LIN {X 0,Y 183.48,Z 465.973,A -85,B 0,C 180,E1 -22041.184,E2 -22041.184} C_VEL
LIN {X 0,Y 183.189,Z 466.318,A -85,B 0,C 180,E1 -22045.596,E2 -22045.596} C_VEL
LIN {X 0,Y 183.308,Z 465.887,A -85,B 0,C 180,E1 -22047.799,E2 -22047.799} C_VEL
LIN {X 0,Y 183.482,Z 465.038,A -85,B 0,C 180,E1 -22049.996,E2 -22049.996} C_VEL
LIN {X 0,Y 183.338,Z 463.763,A -85,B 0,C 180,E1 -22052.193,E2 -22052.193} C_VEL
LIN {X 0,Y 183.267,Z 461.02,A -85,B 0,C 180,E1 -22055.497,E2 -22055.497} C_VEL
LIN {X 0,Y 183.529,Z 457.223,A -85,B 0,C 180,E1 -22058.806,E2 -22058.806} C_VEL
LIN {X 0,Y 184.122,Z 452.262,A -85,B 0,C 180,E1 -22062.114,E2 -22062.114} C_VEL
LIN {X 0,Y 185.268,Z 446.001,A -85,B 0,C 180,E1 -22065.394,E2 -22065.394} C_VEL
LIN {X 0,Y 186.943,Z 438.169,A -85,B 0,C 180,E1 -22068.63,E2 -22068.63} C_VEL
LIN {X 0,Y 188.899,Z 429.24,A -85,B 0,C 180,E1 -22071.543,E2 -22071.543} C_VEL
LIN {X 0,Y 190.919,Z 420.311,A -85,B 0,C 180,E1 -22073.88,E2 -22073.88} C_VEL
LIN {X 0,Y 193.253,Z 409.393,A -85,B 0,C 180,E1 -22076.158,E2 -22076.158} C_VEL
LIN {X 0,Y 195.335,Z 398.733,A -85,B 0,C 180,E1 -22077.88,E2 -22077.88} C_VEL
LIN {X 0,Y 197.244,Z 387.011,A -85,B 0,C 180,E1 -22079.329,E2 -22079.329} C_VEL
LIN {X 0,Y 198.937,Z 373.736,A -85,B 0,C 180,E1 -22080.513,E2 -22080.513} C_VEL
LIN {X 0,Y 199.925,Z 361.7,A -85,B 0,C 180,E1 -22081.225,E2 -22081.225} C_VEL
LIN {X 0,Y 201.881,Z 312.915,A -85,B 0,C 180,E1 -22082.925,E2 -22082.925} C_VEL
LIN {X 0,Y 198.695,Z 281.913,A -85,B 0,C 180,E1 -22084.649,E2 -22084.649} C_VEL
LIN {X 0,Y 191.948,Z 264.141,A -85,B 0,C 180,E1 -22086.507,E2 -22086.507} C_VEL
LIN {X 0,Y 187.121,Z 252.944,A -85,B 0,C 180,E1 -22087.932,E2 -22087.932} C_VEL
LIN {X 0,Y 185.488,Z 246.381,A -85,B 0,C 180,E1 -22091.468,E2 -22091.468} C_VEL
LIN {X 0,Y 185.505,Z 246.376,A -85,B 0,C 180,E1 -22097.003,E2 -22097.003} C_VEL
LIN {X 0,Y 185.519,Z 246.373,A -85,B 0,C 180,E1 -22099.908,E2 -22099.908} C_VEL
LIN {X 0,Y 185.525,Z 246.373,A -85,B 0,C 180,E1 -22102.691,E2 -22102.691} C_VEL
LIN {X 0,Y 185.521,Z 246.373,A -85,B 0,C 180,E1 -22107.97,E2 -22107.97} C_VEL
LIN {X 0,Y 185.559,Z 246.367,A -85,B 0,C 180,E1 -22110.572,E2 -22110.572} C_VEL
LIN {X 0,Y 185.583,Z 246.364,A -85,B 0,C 180,E1 -22115.381,E2 -22115.381} C_VEL
LIN {X 0,Y 185.685,Z 246.348,A -85,B 0,C 180,E1 -22121.098,E2 -22121.098} C_VEL
LIN {X 0,Y 185.696,Z 246.35,A -85,B 0,C 180,E1 -22126.874,E2 -22126.874} C_VEL
LIN {X 0,Y 185.978,Z 246.319,A -85,B 0,C 180,E1 -22131.305,E2 -22131.305} C_VEL
LIN {X 0,Y 186.171,Z 246.257,A -85,B 0,C 180,E1 -22137.836,E2 -22137.836} C_VEL
LIN {X 0,Y 186.367,Z 246.222,A -85,B 0,C 180,E1 -22139.999,E2 -22139.999} C_VEL
LIN {X 0,Y 185.874,Z 246.321,A -85,B 0,C 180,E1 -22144.336,E2 -22144.336} C_VEL
LIN {X 0,Y 185.944,Z 246.321,A -85,B 0,C 180,E1 -22148.695,E2 -22148.695} C_VEL
LIN {X 0,Y 185.684,Z 246.349,A -85,B 0,C 180,E1 -22153.125,E2 -22153.125} C_VEL
LIN {X 0,Y 185.621,Z 246.358,A -85,B 0,C 180,E1 -22157.631,E2 -22157.631} C_VEL
LIN {X 0,Y 185.524,Z 246.372,A -85,B 0,C 180,E1 -22162.26,E2 -22162.26} C_VEL
LIN {X 0,Y 185.552,Z 246.369,A -85,B 0,C 180,E1 -22164.649,E2 -22164.649} C_VEL
LIN {X 0,Y 185.491,Z 246.34,A -85,B 0,C 180,E1 -22169.508,E2 -22169.508} C_VEL
LIN {X 0,Y 185.504,Z 246.357,A -85,B 0,C 180,E1 -22173.556,E2 -22173.556} C_VEL
LIN {X 0,Y 185.478,Z 246.379,A -85,B 0,C 180,E1 -22177.319,E2 -22177.319} C_VEL
LIN {X 0,Y 185.442,Z 246.369,A -85,B 0,C 180,E1 -22180.726,E2 -22180.726} C_VEL
LIN {X 0,Y 185.438,Z 246.378,A -85,B 0,C 180,E1 -22186.061,E2 -22186.061} C_VEL
LIN {X 0,Y 185.442,Z 246.38,A -85,B 0,C 180,E1 -22189.898,E2 -22189.898} C_VEL
LIN {X 0,Y 185.485,Z 246.361,A -85,B 0,C 180,E1 -22192.719,E2 -22192.719} C_VEL
LIN {X 0,Y 185.529,Z 246.368,A -85,B 0,C 180,E1 -22197.98,E2 -22197.98} C_VEL
LIN {X 0,Y 185.569,Z 246.359,A -85,B 0,C 180,E1 -22200.582,E2 -22200.582} C_VEL
LIN {X 0,Y 185.571,Z 246.37,A -85,B 0,C 180,E1 -22205.387,E2 -22205.387} C_VEL
LIN {X 0,Y 185.609,Z 246.365,A -85,B 0,C 180,E1 -22207.242,E2 -22207.242} C_VEL
LIN {X 0,Y 186.764,Z 249.452,A -85,B 0,C 180,E1 -22207.644,E2 -22207.644} C_VEL
LIN {X 0,Y 194.117,Z 263.081,A -85,B 0,C 180,E1 -22209.558,E2 -22209.558} C_VEL
LIN {X 0,Y 200.763,Z 277.43,A -85,B 0,C 180,E1 -22211.227,E2 -22211.227} C_VEL
LIN {X 0,Y 203.132,Z 283.452,A -85,B 0,C 180,E1 -22211.825,E2 -22211.825} C_VEL
LIN {X 0,Y 200.223,Z 346.141,A -85,B 0,C 180,E1 -22213.959,E2 -22213.959} C_VEL
LIN {X 0,Y 199.136,Z 359.93,A -85,B 0,C 180,E1 -22214.853,E2 -22214.853} C_VEL
LIN {X 0,Y 197.648,Z 372.862,A -85,B 0,C 180,E1 -22216.117,E2 -22216.117} C_VEL
LIN {X 0,Y 195.686,Z 385.45,A -85,B 0,C 180,E1 -22217.824,E2 -22217.824} C_VEL
LIN {X 0,Y 193.672,Z 396.651,A -85,B 0,C 180,E1 -22219.815,E2 -22219.815} C_VEL
LIN {X 0,Y 191.332,Z 407.537,A -85,B 0,C 180,E1 -22222.298,E2 -22222.298} C_VEL
LIN {X 0,Y 189.051,Z 417.525,A -85,B 0,C 180,E1 -22225.206,E2 -22225.206} C_VEL
LIN {X 0,Y 187.057,Z 426.077,A -85,B 0,C 180,E1 -22228.389,E2 -22228.389} C_VEL
LIN {X 0,Y 185.529,Z 432.936,A -85,B 0,C 180,E1 -22231.632,E2 -22231.632} C_VEL
LIN {X 0,Y 184.28,Z 439.243,A -85,B 0,C 180,E1 -22235.474,E2 -22235.474} C_VEL
LIN {X 0,Y 183.521,Z 443.364,A -85,B 0,C 180,E1 -22238.814,E2 -22238.814} C_VEL
LIN {X 0,Y 183.177,Z 445.497,A -85,B 0,C 180,E1 -22241.063,E2 -22241.063} C_VEL
LIN {X 0,Y 183.003,Z 447.197,A -85,B 0,C 180,E1 -22243.325,E2 -22243.325} C_VEL
LIN {X 0,Y 183.074,Z 448.781,A -85,B 0,C 180,E1 -22246.32,E2 -22246.32} C_VEL
LIN {X 0,Y 183.511,Z 449.733,A -85,B 0,C 180,E1 -22250.164,E2 -22250.164} C_VEL
LIN {X 0,Y 184.562,Z 449.504,A -85,B 0,C 180,E1 -22253.951,E2 -22253.951} C_VEL
LIN {X 0,Y 185.803,Z 448.458,A -85,B 0,C 180,E1 -22256.996,E2 -22256.996} C_VEL
LIN {X 0,Y 187.881,Z 446.113,A -85,B 0,C 180,E1 -22260.645,E2 -22260.645} C_VEL
LIN {X 0,Y 190.154,Z 443.163,A -85,B 0,C 180,E1 -22263.67,E2 -22263.67} C_VEL
LIN {X 0,Y 192.997,Z 439.038,A -85,B 0,C 180,E1 -22266.763,E2 -22266.763} C_VEL
LIN {X 0,Y 196.675,Z 433.185,A -85,B 0,C 180,E1 -22270.032,E2 -22270.032} C_VEL
LIN {X 0,Y 200.751,Z 425.989,A -85,B 0,C 180,E1 -22273.082,E2 -22273.082} C_VEL
LIN {X 0,Y 204.49,Z 418.653,A -85,B 0,C 180,E1 -22275.491,E2 -22275.491} C_VEL
LIN {X 0,Y 209.025,Z 408.565,A -85,B 0,C 180,E1 -22278.064,E2 -22278.064} C_VEL
LIN {X 0,Y 213.085,Z 398.325,A -85,B 0,C 180,E1 -22280.069,E2 -22280.069} C_VEL
LIN {X 0,Y 216.691,Z 387.306,A -85,B 0,C 180,E1 -22281.743,E2 -22281.743} C_VEL
LIN {X 0,Y 219.669,Z 375.741,A -85,B 0,C 180,E1 -22283.113,E2 -22283.113} C_VEL
LIN {X 0,Y 222.119,Z 363.633,A -85,B 0,C 180,E1 -22284.172,E2 -22284.172} C_VEL
LIN {X 0,Y 223.883,Z 351.06,A -85,B 0,C 180,E1 -22284.937,E2 -22284.937} C_VEL
LIN {X 0,Y 225.127,Z 335.128,A -85,B 0,C 180,E1 -22285.509,E2 -22285.509} C_VEL
LIN {X 0,Y 227.022,Z 306.267,A -85,B 0,C 180,E1 -22286.336,E2 -22286.336} C_VEL
LIN {X 0,Y 222.883,Z 298.122,A -85,B 0,C 180,E1 -22287.919,E2 -22287.919} C_VEL
LIN {X 0,Y 216.346,Z 287.146,A -85,B 0,C 180,E1 -22290.572,E2 -22290.572} C_VEL
LIN {X 0,Y 210.785,Z 278.967,A -85,B 0,C 180,E1 -22293.05,E2 -22293.05} C_VEL
LIN {X 0,Y 207.966,Z 274.951,A -85,B 0,C 180,E1 -22294.411,E2 -22294.411} C_VEL
LIN {X 0,Y 205.236,Z 271.19,A -85,B 0,C 180,E1 -22295.805,E2 -22295.805} C_VEL
LIN {X 0,Y 202.511,Z 267.488,A -85,B 0,C 180,E1 -22297.289,E2 -22297.289} C_VEL
LIN {X 0,Y 199.691,Z 263.918,A -85,B 0,C 180,E1 -22298.922,E2 -22298.922} C_VEL
LIN {X 0,Y 198.86,Z 262.779,A -85,B 0,C 180,E1 -22299.44,E2 -22299.44} C_VEL
LIN {X 0,Y 196.208,Z 259.92,A -85,B 0,C 180,E1 -22301.126,E2 -22301.126} C_VEL
LIN {X 0,Y 194.881,Z 257.667,A -85,B 0,C 180,E1 -22302.096,E2 -22302.096} C_VEL
LIN {X 0,Y 192.271,Z 255.408,A -85,B 0,C 180,E1 -22303.954,E2 -22303.954} C_VEL
LIN {X 0,Y 190.705,Z 252.456,A -85,B 0,C 180,E1 -22305.324,E2 -22305.324} C_VEL
LIN {X 0,Y 187.601,Z 250.288,A -85,B 0,C 180,E1 -22307.973,E2 -22307.973} C_VEL
LIN {X 0,Y 186.312,Z 248.073,A -85,B 0,C 180,E1 -22309.376,E2 -22309.376} C_VEL
LIN {X 0,Y 185.892,Z 246.326,A -85,B 0,C 180,E1 -22310.072,E2 -22310.072} C_VEL
LIN {X 0,Y 185.931,Z 246.315,A -85,B 0,C 180,E1 -22313.49,E2 -22313.49} C_VEL
LIN {X 0,Y 186.191,Z 246.277,A -85,B 0,C 180,E1 -22317.837,E2 -22317.837} C_VEL
LIN {X 0,Y 186.388,Z 246.25,A -85,B 0,C 180,E1 -22320.001,E2 -22320.001} C_VEL
LIN {X 0,Y 185.89,Z 246.314,A -85,B 0,C 180,E1 -22324.337,E2 -22324.337} C_VEL
LIN {X 0,Y 185.964,Z 246.308,A -85,B 0,C 180,E1 -22328.695,E2 -22328.695} C_VEL
LIN {X 0,Y 185.696,Z 246.344,A -85,B 0,C 180,E1 -22333.126,E2 -22333.126} C_VEL
LIN {X 0,Y 185.621,Z 246.348,A -85,B 0,C 180,E1 -22338.821,E2 -22338.821} C_VEL
LIN {X 0,Y 185.546,Z 246.398,A -85,B 0,C 180,E1 -22341.966,E2 -22341.966} C_VEL
LIN {X 0,Y 186.271,Z 248.742,A -85,B 0,C 180,E1 -22345.086,E2 -22345.086} C_VEL
LIN {X 0,Y 191.23,Z 255.196,A -85,B 0,C 180,E1 -22349.734,E2 -22349.734} C_VEL
LIN {X 0,Y 192.349,Z 256.695,A -85,B 0,C 180,E1 -22350.632,E2 -22350.632} C_VEL
LIN {X 0,Y 196.512,Z 262.285,A -85,B 0,C 180,E1 -22353.654,E2 -22353.654} C_VEL
LIN {X 0,Y 201.46,Z 269.683,A -85,B 0,C 180,E1 -22356.781,E2 -22356.781} C_VEL
LIN {X 0,Y 205.46,Z 275.971,A -85,B 0,C 180,E1 -22359.019,E2 -22359.019} C_VEL
LIN {X 0,Y 209.158,Z 282.09,A -85,B 0,C 180,E1 -22360.923,E2 -22360.923} C_VEL
LIN {X 0,Y 213.972,Z 290.647,A -85,B 0,C 180,E1 -22363.213,E2 -22363.213} C_VEL
LIN {X 0,Y 219.624,Z 301.889,A -85,B 0,C 180,E1 -22365.689,E2 -22365.689} C_VEL
LIN {X 0,Y 225.322,Z 315.327,A -85,B 0,C 180,E1 -22368.033,E2 -22368.033} C_VEL
LIN {X 0,Y 226.072,Z 322.786,A -85,B 0,C 180,E1 -22368.592,E2 -22368.592} C_VEL
LIN {X 0,Y 224.889,Z 341.991,A -85,B 0,C 180,E1 -22369.163,E2 -22369.163} C_VEL
LIN {X 0,Y 224.046,Z 347.848,A -85,B 0,C 180,E1 -22369.2,E2 -22369.2} C_VEL
LIN {X 0,Y 219.07,Z 364.929,A -85,B 0,C 180,E1 -22368.799,E2 -22368.799} C_VEL
LIN {X 0,Y 217.556,Z 370.627,A -85,B 0,C 180,E1 -22368.885,E2 -22368.885} C_VEL
LIN {X 0,Y 217.166,Z 372.524,A -85,B 0,C 180,E1 -22368.977,E2 -22368.977} C_VEL
LIN {X 0,Y 214.578,Z 385.014,A -85,B 0,C 180,E1 -22369.848,E2 -22369.848} C_VEL
LIN {X 0,Y 211.184,Z 397.55,A -85,B 0,C 180,E1 -22371.087,E2 -22371.087} C_VEL
LIN {X 0,Y 207.117,Z 409.31,A -85,B 0,C 180,E1 -22372.66,E2 -22372.66} C_VEL
LIN {X 0,Y 202.865,Z 419.845,A -85,B 0,C 180,E1 -22374.529,E2 -22374.529} C_VEL
LIN {X 0,Y 198.429,Z 429.37,A -85,B 0,C 180,E1 -22376.702,E2 -22376.702} C_VEL
LIN {X 0,Y 193.641,Z 438.575,A -85,B 0,C 180,E1 -22379.461,E2 -22379.461} C_VEL
LIN {X 0,Y 189.347,Z 446.004,A -85,B 0,C 180,E1 -22382.356,E2 -22382.356} C_VEL
LIN {X 0,Y 185.796,Z 452.003,A -85,B 0,C 180,E1 -22385.41,E2 -22385.41} C_VEL
LIN {X 0,Y 182.64,Z 456.782,A -85,B 0,C 180,E1 -22388.556,E2 -22388.556} C_VEL
LIN {X 0,Y 180.104,Z 460.476,A -85,B 0,C 180,E1 -22391.807,E2 -22391.807} C_VEL
LIN {X 0,Y 178.696,Z 462.406,A -85,B 0,C 180,E1 -22394.017,E2 -22394.017} C_VEL
LIN {X 0,Y 177.692,Z 463.905,A -85,B 0,C 180,E1 -22396.269,E2 -22396.269} C_VEL
LIN {X 0,Y 176.442,Z 465.693,A -85,B 0,C 180,E1 -22400.829,E2 -22400.829} C_VEL
LIN {X 0,Y 176.111,Z 465.962,A -85,B 0,C 180,E1 -22405.419,E2 -22405.419} C_VEL
LIN {X 0,Y 176.225,Z 465.477,A -85,B 0,C 180,E1 -22407.711,E2 -22407.711} C_VEL
LIN {X 0,Y 176.394,Z 464.596,A -85,B 0,C 180,E1 -22409.996,E2 -22409.996} C_VEL
LIN {X 0,Y 176.182,Z 461.827,A -85,B 0,C 180,E1 -22414.23,E2 -22414.23} C_VEL
LIN {X 0,Y 176.37,Z 458.041,A -85,B 0,C 180,E1 -22418.012,E2 -22418.012} C_VEL
LIN {X 0,Y 176.861,Z 453.396,A -85,B 0,C 180,E1 -22421.455,E2 -22421.455} C_VEL
LIN {X 0,Y 178.124,Z 446.34,A -85,B 0,C 180,E1 -22425.44,E2 -22425.44} C_VEL
LIN {X 0,Y 179.813,Z 438.686,A -85,B 0,C 180,E1 -22428.805,E2 -22428.805} C_VEL
LIN {X 0,Y 181.124,Z 432.844,A -85,B 0,C 180,E1 -22430.903,E2 -22430.903} C_VEL
LIN {X 0,Y 183.516,Z 423.354,A -85,B 0,C 180,E1 -22433.704,E2 -22433.704} C_VEL
LIN {X 0,Y 185.65,Z 413.191,A -85,B 0,C 180,E1 -22436.102,E2 -22436.102} C_VEL
LIN {X 0,Y 188.02,Z 401.911,A -85,B 0,C 180,E1 -22438.151,E2 -22438.151} C_VEL
LIN {X 0,Y 189.81,Z 392.258,A -85,B 0,C 180,E1 -22439.525,E2 -22439.525} C_VEL
LIN {X 0,Y 191.695,Z 379.731,A -85,B 0,C 180,E1 -22440.875,E2 -22440.875} C_VEL
LIN {X 0,Y 193.052,Z 367.735,A -85,B 0,C 180,E1 -22441.777,E2 -22441.777} C_VEL
LIN {X 0,Y 193.951,Z 354.677,A -85,B 0,C 180,E1 -22442.378,E2 -22442.378} C_VEL
LIN {X 0,Y 195.524,Z 313.461,A -85,B 0,C 180,E1 -22443.841,E2 -22443.841} C_VEL
LIN {X 0,Y 192.584,Z 283.99,A -85,B 0,C 180,E1 -22445.547,E2 -22445.547} C_VEL
LIN {X 0,Y 185.649,Z 265.778,A -85,B 0,C 180,E1 -22447.568,E2 -22447.568} C_VEL
LIN {X 0,Y 180.831,Z 255.242,A -85,B 0,C 180,E1 -22448.985,E2 -22448.985} C_VEL
LIN {X 0,Y 179.766,Z 252.638,A -85,B 0,C 180,E1 -22449.355,E2 -22449.355} C_VEL
LIN {X 0,Y 178.435,Z 247.258,A -85,B 0,C 180,E1 -22452.405,E2 -22452.405} C_VEL
LIN {X 0,Y 178.43,Z 247.258,A -85,B 0,C 180,E1 -22457.963,E2 -22457.963} C_VEL
LIN {X 0,Y 178.455,Z 247.256,A -85,B 0,C 180,E1 -22461.953,E2 -22461.953} C_VEL
LIN {X 0,Y 178.467,Z 247.25,A -85,B 0,C 180,E1 -22466.542,E2 -22466.542} C_VEL
LIN {X 0,Y 178.5,Z 247.247,A -85,B 0,C 180,E1 -22470.002,E2 -22470.002} C_VEL
LIN {X 0,Y 178.511,Z 247.247,A -85,B 0,C 180,E1 -22474.872,E2 -22474.872} C_VEL
LIN {X 0,Y 178.629,Z 247.228,A -85,B 0,C 180,E1 -22480.752,E2 -22480.752} C_VEL
LIN {X 0,Y 178.625,Z 247.232,A -85,B 0,C 180,E1 -22486.345,E2 -22486.345} C_VEL
LIN {X 0,Y 178.908,Z 247.197,A -85,B 0,C 180,E1 -22490.959,E2 -22490.959} C_VEL
LIN {X 0,Y 179.117,Z 247.134,A -85,B 0,C 180,E1 -22497.751,E2 -22497.751} C_VEL
LIN {X 0,Y 179.33,Z 247.096,A -85,B 0,C 180,E1 -22499.999,E2 -22499.999} C_VEL
LIN {X 0,Y 178.822,Z 247.199,A -85,B 0,C 180,E1 -22504.508,E2 -22504.508} C_VEL
LIN {X 0,Y 178.875,Z 247.199,A -85,B 0,C 180,E1 -22509.041,E2 -22509.041} C_VEL
LIN {X 0,Y 178.61,Z 247.234,A -85,B 0,C 180,E1 -22513.655,E2 -22513.655} C_VEL
LIN {X 0,Y 178.526,Z 247.234,A -85,B 0,C 180,E1 -22519.152,E2 -22519.152} C_VEL
LIN {X 0,Y 178.49,Z 247.246,A -85,B 0,C 180,E1 -22525.114,E2 -22525.114} C_VEL
LIN {X 0,Y 178.425,Z 247.213,A -85,B 0,C 180,E1 -22530.8,E2 -22530.8} C_VEL
LIN {X 0,Y 178.459,Z 247.24,A -85,B 0,C 180,E1 -22534.222,E2 -22534.222} C_VEL
LIN {X 0,Y 178.367,Z 247.26,A -85,B 0,C 180,E1 -22539.081,E2 -22539.081} C_VEL
LIN {X 0,Y 178.374,Z 247.236,A -85,B 0,C 180,E1 -22542.051,E2 -22542.051} C_VEL
LIN {X 0,Y 178.373,Z 247.248,A -85,B 0,C 180,E1 -22545.17,E2 -22545.17} C_VEL
LIN {X 0,Y 178.382,Z 247.265,A -85,B 0,C 180,E1 -22548.466,E2 -22548.466} C_VEL
LIN {X 0,Y 178.404,Z 247.248,A -85,B 0,C 180,E1 -22553.787,E2 -22553.787} C_VEL
LIN {X 0,Y 178.472,Z 247.254,A -85,B 0,C 180,E1 -22556.552,E2 -22556.552} C_VEL
LIN {X 0,Y 178.51,Z 247.235,A -85,B 0,C 180,E1 -22560.013,E2 -22560.013} C_VEL
LIN {X 0,Y 178.564,Z 247.3,A -85,B 0,C 180,E1 -22565.904,E2 -22565.904} C_VEL
LIN {X 0,Y 179.536,Z 250.057,A -85,B 0,C 180,E1 -22566.24,E2 -22566.24} C_VEL
LIN {X 0,Y 180.838,Z 252.082,A -85,B 0,C 180,E1 -22566.603,E2 -22566.603} C_VEL
LIN {X 0,Y 189.565,Z 268.477,A -85,B 0,C 180,E1 -22568.999,E2 -22568.999} C_VEL
LIN {X 0,Y 196.436,Z 284.081,A -85,B 0,C 180,E1 -22570.823,E2 -22570.823} C_VEL
LIN {X 0,Y 196.814,Z 285.071,A -85,B 0,C 180,E1 -22570.924,E2 -22570.924} C_VEL
LIN {X 0,Y 193.783,Z 346.955,A -85,B 0,C 180,E1 -22573.091,E2 -22573.091} C_VEL
LIN {X 0,Y 192.685,Z 360.358,A -85,B 0,C 180,E1 -22573.994,E2 -22573.994} C_VEL
LIN {X 0,Y 191.21,Z 372.74,A -85,B 0,C 180,E1 -22575.232,E2 -22575.232} C_VEL
LIN {X 0,Y 189.33,Z 384.629,A -85,B 0,C 180,E1 -22576.863,E2 -22576.863} C_VEL
LIN {X 0,Y 187.159,Z 396.054,A -85,B 0,C 180,E1 -22578.909,E2 -22578.909} C_VEL
LIN {X 0,Y 184.961,Z 406.355,A -85,B 0,C 180,E1 -22581.262,E2 -22581.262} C_VEL
LIN {X 0,Y 182.737,Z 415.618,A -85,B 0,C 180,E1 -22583.933,E2 -22583.933} C_VEL
LIN {X 0,Y 180.518,Z 424.625,A -85,B 0,C 180,E1 -22587.215,E2 -22587.215} C_VEL
LIN {X 0,Y 178.814,Z 431.868,A -85,B 0,C 180,E1 -22590.567,E2 -22590.567} C_VEL
LIN {X 0,Y 177.743,Z 436.756,A -85,B 0,C 180,E1 -22593.404,E2 -22593.404} C_VEL
LIN {X 0,Y 176.823,Z 441.511,A -85,B 0,C 180,E1 -22596.851,E2 -22596.851} C_VEL
LIN {X 0,Y 176.162,Z 445.159,A -85,B 0,C 180,E1 -22600.345,E2 -22600.345} C_VEL
LIN {X 0,Y 175.909,Z 447.771,A -85,B 0,C 180,E1 -22603.872,E2 -22603.872} C_VEL
LIN {X 0,Y 175.988,Z 449.101,A -85,B 0,C 180,E1 -22606.581,E2 -22606.581} C_VEL
LIN {X 0,Y 176.575,Z 450.1,A -85,B 0,C 180,E1 -22610.993,E2 -22610.993} C_VEL
LIN {X 0,Y 177.615,Z 449.849,A -85,B 0,C 180,E1 -22614.485,E2 -22614.485} C_VEL
LIN {X 0,Y 179.177,Z 448.61,A -85,B 0,C 180,E1 -22618.08,E2 -22618.08} C_VEL
LIN {X 0,Y 181.188,Z 446.488,A -85,B 0,C 180,E1 -22621.424,E2 -22621.424} C_VEL
LIN {X 0,Y 183.957,Z 443.085,A -85,B 0,C 180,E1 -22624.965,E2 -22624.965} C_VEL
LIN {X 0,Y 187.263,Z 438.537,A -85,B 0,C 180,E1 -22628.329,E2 -22628.329} C_VEL
LIN {X 0,Y 191.022,Z 432.847,A -85,B 0,C 180,E1 -22631.472,E2 -22631.472} C_VEL
LIN {X 0,Y 195.368,Z 425.496,A -85,B 0,C 180,E1 -22634.545,E2 -22634.545} C_VEL
LIN {X 0,Y 199.33,Z 417.91,A -85,B 0,C 180,E1 -22637.021,E2 -22637.021} C_VEL
LIN {X 0,Y 203.692,Z 408.636,A -85,B 0,C 180,E1 -22639.381,E2 -22639.381} C_VEL
LIN {X 0,Y 207.907,Z 398.332,A -85,B 0,C 180,E1 -22641.416,E2 -22641.416} C_VEL
LIN {X 0,Y 211.769,Z 386.84,A -85,B 0,C 180,E1 -22643.156,E2 -22643.156} C_VEL
LIN {X 0,Y 214.764,Z 375.478,A -85,B 0,C 180,E1 -22644.499,E2 -22644.499} C_VEL
LIN {X 0,Y 217.314,Z 363.255,A -85,B 0,C 180,E1 -22645.554,E2 -22645.554} C_VEL
LIN {X 0,Y 219.098,Z 350.68,A -85,B 0,C 180,E1 -22646.301,E2 -22646.301} C_VEL
LIN {X 0,Y 220.542,Z 332.302,A -85,B 0,C 180,E1 -22646.934,E2 -22646.934} C_VEL
LIN {X 0,Y 222.045,Z 308.741,A -85,B 0,C 180,E1 -22647.646,E2 -22647.646} C_VEL
LIN {X 0,Y 216.6,Z 298.559,A -85,B 0,C 180,E1 -22649.874,E2 -22649.874} C_VEL
LIN {X 0,Y 210.811,Z 289.122,A -85,B 0,C 180,E1 -22652.448,E2 -22652.448} C_VEL
LIN {X 0,Y 205.424,Z 281.137,A -85,B 0,C 180,E1 -22655.088,E2 -22655.088} C_VEL
LIN {X 0,Y 202.251,Z 276.704,A -85,B 0,C 180,E1 -22656.786,E2 -22656.786} C_VEL
LIN {X 0,Y 199.894,Z 273.49,A -85,B 0,C 180,E1 -22658.133,E2 -22658.133} C_VEL
LIN {X 0,Y 197.095,Z 269.678,A -85,B 0,C 180,E1 -22659.86,E2 -22659.86} C_VEL
LIN {X 0,Y 193.782,Z 265.758,A -85,B 0,C 180,E1 -22662.08,E2 -22662.08} C_VEL
LIN {X 0,Y 192.836,Z 264.17,A -85,B 0,C 180,E1 -22662.803,E2 -22662.803} C_VEL
LIN {X 0,Y 190.258,Z 261.653,A -85,B 0,C 180,E1 -22664.758,E2 -22664.758} C_VEL
LIN {X 0,Y 188.591,Z 258.894,A -85,B 0,C 180,E1 -22666.258,E2 -22666.258} C_VEL
LIN {X 0,Y 185.916,Z 256.777,A -85,B 0,C 180,E1 -22668.692,E2 -22668.692} C_VEL
LIN {X 0,Y 184.495,Z 254.18,A -85,B 0,C 180,E1 -22670.351,E2 -22670.351} C_VEL
LIN {X 0,Y 184.119,Z 253.176,A -85,B 0,C 180,E1 -22670.863,E2 -22670.863} C_VEL
LIN {X 0,Y 180.894,Z 251.356,A -85,B 0,C 180,E1 -22674.986,E2 -22674.986} C_VEL
LIN {X 0,Y 179.646,Z 249.237,A -85,B 0,C 180,E1 -22677.408,E2 -22677.408} C_VEL
LIN {X 0,Y 179.217,Z 247.155,A -85,B 0,C 180,E1 -22678.877,E2 -22678.877} C_VEL
LIN {X 0,Y 179.352,Z 247.126,A -85,B 0,C 180,E1 -22680.001,E2 -22680.001} C_VEL
LIN {X 0,Y 178.838,Z 247.19,A -85,B 0,C 180,E1 -22684.509,E2 -22684.509} C_VEL
LIN {X 0,Y 178.896,Z 247.184,A -85,B 0,C 180,E1 -22689.042,E2 -22689.042} C_VEL
LIN {X 0,Y 178.626,Z 247.351,A -85,B 0,C 180,E1 -22694.381,E2 -22694.381} C_VEL
LIN {X 0,Y 179.442,Z 249.866,A -85,B 0,C 180,E1 -22696.79,E2 -22696.79} C_VEL
LIN {X 0,Y 182.102,Z 252.583,A -85,B 0,C 180,E1 -22701.213,E2 -22701.213} C_VEL
LIN {X 0,Y 184.513,Z 255.018,A -85,B 0,C 180,E1 -22704.194,E2 -22704.194} C_VEL
LIN {X 0,Y 189.564,Z 261.854,A -85,B 0,C 180,E1 -22709.187,E2 -22709.187} C_VEL
LIN {X 0,Y 194.945,Z 269.613,A -85,B 0,C 180,E1 -22713.347,E2 -22713.347} C_VEL
LIN {X 0,Y 198.956,Z 275.781,A -85,B 0,C 180,E1 -22715.982,E2 -22715.982} C_VEL
LIN {X 0,Y 202.623,Z 281.711,A -85,B 0,C 180,E1 -22718.139,E2 -22718.139} C_VEL
LIN {X 0,Y 207.617,Z 290.164,A -85,B 0,C 180,E1 -22720.795,E2 -22720.795} C_VEL
LIN {X 0,Y 213.536,Z 301.679,A -85,B 0,C 180,E1 -22723.668,E2 -22723.668} C_VEL
LIN {X 0,Y 218.355,Z 312.563,A -85,B 0,C 180,E1 -22725.836,E2 -22725.836} C_VEL
LIN {X 0,Y 220.759,Z 318.702,A -85,B 0,C 180,E1 -22726.878,E2 -22726.878} C_VEL
LIN {X 0,Y 221.199,Z 324.248,A -85,B 0,C 180,E1 -22727.28,E2 -22727.28} C_VEL
LIN {X 0,Y 218.625,Z 361.808,A -85,B 0,C 180,E1 -22728.449,E2 -22728.449} C_VEL
LIN {X 0,Y 217.166,Z 372.524,A -85,B 0,C 180,E1 -22728.977,E2 -22728.977} C_VEL
LIN {X 0,Y 214.834,Z 379.991,A -85,B 0,C 180,E1 -22729.217,E2 -22729.217} C_VEL
LIN {X 0,Y 211.413,Z 387.173,A -85,B 0,C 180,E1 -22729.304,E2 -22729.304} C_VEL
LIN {X 0,Y 207.012,Z 395.981,A -85,B 0,C 180,E1 -22729.663,E2 -22729.663} C_VEL
LIN {X 0,Y 204.895,Z 401.136,A -85,B 0,C 180,E1 -22730.166,E2 -22730.166} C_VEL
LIN {X 0,Y 200.526,Z 412.62,A -85,B 0,C 180,E1 -22731.85,E2 -22731.85} C_VEL
LIN {X 0,Y 196.169,Z 422.449,A -85,B 0,C 180,E1 -22733.762,E2 -22733.762} C_VEL
LIN {X 0,Y 191.693,Z 431.406,A -85,B 0,C 180,E1 -22736.005,E2 -22736.005} C_VEL
LIN {X 0,Y 186.768,Z 440.184,A -85,B 0,C 180,E1 -22738.84,E2 -22738.84} C_VEL
LIN {X 0,Y 182.406,Z 447.248,A -85,B 0,C 180,E1 -22741.835,E2 -22741.835} C_VEL
LIN {X 0,Y 178.205,Z 453.735,A -85,B 0,C 180,E1 -22745.536,E2 -22745.536} C_VEL
LIN {X 0,Y 175.056,Z 458.059,A -85,B 0,C 180,E1 -22748.816,E2 -22748.816} C_VEL
LIN {X 0,Y 173.359,Z 460.369,A -85,B 0,C 180,E1 -22751.073,E2 -22751.073} C_VEL
LIN {X 0,Y 171.86,Z 462.254,A -85,B 0,C 180,E1 -22753.363,E2 -22753.363} C_VEL
LIN {X 0,Y 169.982,Z 464.743,A -85,B 0,C 180,E1 -22758.066,E2 -22758.066} C_VEL
LIN {X 0,Y 169.089,Z 465.708,A -85,B 0,C 180,E1 -22762.834,E2 -22762.834} C_VEL
LIN {X 0,Y 169.043,Z 465.413,A -85,B 0,C 180,E1 -22766.212,E2 -22766.212} C_VEL
LIN {X 0,Y 169.309,Z 464.151,A -85,B 0,C 180,E1 -22769.996,E2 -22769.996} C_VEL
LIN {X 0,Y 169.102,Z 461.559,A -85,B 0,C 180,E1 -22774.078,E2 -22774.078} C_VEL
LIN {X 0,Y 169.307,Z 457.418,A -85,B 0,C 180,E1 -22778.349,E2 -22778.349} C_VEL
LIN {X 0,Y 169.862,Z 452.687,A -85,B 0,C 180,E1 -22781.934,E2 -22781.934} C_VEL
LIN {X 0,Y 171.008,Z 446.676,A -85,B 0,C 180,E1 -22785.488,E2 -22785.488} C_VEL
LIN {X 0,Y 172.691,Z 439.16,A -85,B 0,C 180,E1 -22788.994,E2 -22788.994} C_VEL
LIN {X 0,Y 174.143,Z 433.136,A -85,B 0,C 180,E1 -22791.292,E2 -22791.292} C_VEL
LIN {X 0,Y 176.477,Z 424.18,A -85,B 0,C 180,E1 -22794.085,E2 -22794.085} C_VEL
LIN {X 0,Y 178.714,Z 414.288,A -85,B 0,C 180,E1 -22796.565,E2 -22796.565} C_VEL
LIN {X 0,Y 181.08,Z 403.438,A -85,B 0,C 180,E1 -22798.697,E2 -22798.697} C_VEL
LIN {X 0,Y 183.125,Z 393.27,A -85,B 0,C 180,E1 -22800.239,E2 -22800.239} C_VEL
LIN {X 0,Y 185.081,Z 381.159,A -85,B 0,C 180,E1 -22801.627,E2 -22801.627} C_VEL
LIN {X 0,Y 186.559,Z 368.94,A -85,B 0,C 180,E1 -22802.62,E2 -22802.62} C_VEL
LIN {X 0,Y 187.593,Z 355.544,A -85,B 0,C 180,E1 -22803.296,E2 -22803.296} C_VEL
LIN {X 0,Y 189.299,Z 314.801,A -85,B 0,C 180,E1 -22804.772,E2 -22804.772} C_VEL
LIN {X 0,Y 186.547,Z 286.215,A -85,B 0,C 180,E1 -22806.493,E2 -22806.493} C_VEL
LIN {X 0,Y 179.81,Z 268.274,A -85,B 0,C 180,E1 -22808.581,E2 -22808.581} C_VEL
LIN {X 0,Y 173.93,Z 255.691,A -85,B 0,C 180,E1 -22810.424,E2 -22810.424} C_VEL
LIN {X 0,Y 172.398,Z 252.228,A -85,B 0,C 180,E1 -22810.978,E2 -22810.978} C_VEL
LIN {X 0,Y 171.42,Z 248.132,A -85,B 0,C 180,E1 -22813.427,E2 -22813.427} C_VEL
LIN {X 0,Y 171.361,Z 248.14,A -85,B 0,C 180,E1 -22818.988,E2 -22818.988} C_VEL
LIN {X 0,Y 171.403,Z 248.134,A -85,B 0,C 180,E1 -22822.044,E2 -22822.044} C_VEL
LIN {X 0,Y 171.386,Z 248.135,A -85,B 0,C 180,E1 -22825.084,E2 -22825.084} C_VEL
LIN {X 0,Y 171.427,Z 248.127,A -85,B 0,C 180,E1 -22830.529,E2 -22830.529} C_VEL
LIN {X 0,Y 171.443,Z 248.124,A -85,B 0,C 180,E1 -22835.799,E2 -22835.799} C_VEL
LIN {X 0,Y 171.585,Z 248.105,A -85,B 0,C 180,E1 -22840.872,E2 -22840.872} C_VEL
LIN {X 0,Y 171.545,Z 248.115,A -85,B 0,C 180,E1 -22845.769,E2 -22845.769} C_VEL
LIN {X 0,Y 171.843,Z 248.076,A -85,B 0,C 180,E1 -22850.584,E2 -22850.584} C_VEL
LIN {X 0,Y 171.782,Z 248.072,A -85,B 0,C 180,E1 -22855.306,E2 -22855.306} C_VEL
LIN {X 0,Y 172.294,Z 247.97,A -85,B 0,C 180,E1 -22859.999,E2 -22859.999} C_VEL
LIN {X 0,Y 171.771,Z 248.078,A -85,B 0,C 180,E1 -22864.693,E2 -22864.693} C_VEL
LIN {X 0,Y 171.814,Z 248.077,A -85,B 0,C 180,E1 -22869.416,E2 -22869.416} C_VEL
LIN {X 0,Y 171.525,Z 248.117,A -85,B 0,C 180,E1 -22874.231,E2 -22874.231} C_VEL
LIN {X 0,Y 171.451,Z 248.114,A -85,B 0,C 180,E1 -22879.5,E2 -22879.5} C_VEL
LIN {X 0,Y 171.418,Z 248.126,A -85,B 0,C 180,E1 -22885.6,E2 -22885.6} C_VEL
LIN {X 0,Y 171.38,Z 248.089,A -85,B 0,C 180,E1 -22890.568,E2 -22890.568} C_VEL
LIN {X 0,Y 171.37,Z 248.128,A -85,B 0,C 180,E1 -22895.039,E2 -22895.039} C_VEL
LIN {X 0,Y 171.323,Z 248.139,A -85,B 0,C 180,E1 -22898.806,E2 -22898.806} C_VEL
LIN {X 0,Y 171.3,Z 248.118,A -85,B 0,C 180,E1 -22904.223,E2 -22904.223} C_VEL
LIN {X 0,Y 171.314,Z 248.144,A -85,B 0,C 180,E1 -22908.985,E2 -22908.985} C_VEL
LIN {X 0,Y 171.344,Z 248.12,A -85,B 0,C 180,E1 -22912.039,E2 -22912.039} C_VEL
LIN {X 0,Y 171.384,Z 248.134,A -85,B 0,C 180,E1 -22915.098,E2 -22915.098} C_VEL
LIN {X 0,Y 171.436,Z 248.118,A -85,B 0,C 180,E1 -22920.54,E2 -22920.54} C_VEL
LIN {X 0,Y 171.473,Z 248.213,A -85,B 0,C 180,E1 -22924.38,E2 -22924.38} C_VEL
LIN {X 0,Y 172.442,Z 250.934,A -85,B 0,C 180,E1 -22924.739,E2 -22924.739} C_VEL
LIN {X 0,Y 173.923,Z 253.15,A -85,B 0,C 180,E1 -22925.183,E2 -22925.183} C_VEL
LIN {X 0,Y 182.082,Z 268.126,A -85,B 0,C 180,E1 -22927.598,E2 -22927.598} C_VEL
LIN {X 0,Y 188.603,Z 282.131,A -85,B 0,C 180,E1 -22929.428,E2 -22929.428} C_VEL
LIN {X 0,Y 190.434,Z 286.607,A -85,B 0,C 180,E1 -22929.94,E2 -22929.94} C_VEL
LIN {X 0,Y 187.452,Z 347.231,A -85,B 0,C 180,E1 -22932.137,E2 -22932.137} C_VEL
LIN {X 0,Y 186.279,Z 360.788,A -85,B 0,C 180,E1 -22933.075,E2 -22933.075} C_VEL
LIN {X 0,Y 184.68,Z 373.637,A -85,B 0,C 180,E1 -22934.415,E2 -22934.415} C_VEL
LIN {X 0,Y 182.689,Z 385.409,A -85,B 0,C 180,E1 -22936.093,E2 -22936.093} C_VEL
LIN {X 0,Y 180.453,Z 396.744,A -85,B 0,C 180,E1 -22938.207,E2 -22938.207} C_VEL
LIN {X 0,Y 177.97,Z 407.675,A -85,B 0,C 180,E1 -22940.835,E2 -22940.835} C_VEL
LIN {X 0,Y 175.641,Z 416.995,A -85,B 0,C 180,E1 -22943.687,E2 -22943.687} C_VEL
LIN {X 0,Y 173.39,Z 425.822,A -85,B 0,C 180,E1 -22947.1,E2 -22947.1} C_VEL
LIN {X 0,Y 171.641,Z 432.859,A -85,B 0,C 180,E1 -22950.591,E2 -22950.591} C_VEL
LIN {X 0,Y 170.253,Z 439.309,A -85,B 0,C 180,E1 -22954.739,E2 -22954.739} C_VEL
LIN {X 0,Y 169.399,Z 443.568,A -85,B 0,C 180,E1 -22958.353,E2 -22958.353} C_VEL
LIN {X 0,Y 168.873,Z 446.756,A -85,B 0,C 180,E1 -22962.013,E2 -22962.013} C_VEL
LIN {X 0,Y 168.802,Z 448.336,A -85,B 0,C 180,E1 -22964.469,E2 -22964.469} C_VEL
LIN {X 0,Y 168.925,Z 449.446,A -85,B 0,C 180,E1 -22966.934,E2 -22966.934} C_VEL
LIN {X 0,Y 169.17,Z 450.158,A -85,B 0,C 180,E1 -22969.414,E2 -22969.414} C_VEL
LIN {X 0,Y 169.676,Z 450.466,A -85,B 0,C 180,E1 -22971.89,E2 -22971.89} C_VEL
LIN {X 0,Y 170.698,Z 450.191,A -85,B 0,C 180,E1 -22975.072,E2 -22975.072} C_VEL
LIN {X 0,Y 172.617,Z 448.762,A -85,B 0,C 180,E1 -22979.249,E2 -22979.249} C_VEL
LIN {X 0,Y 174.555,Z 446.855,A -85,B 0,C 180,E1 -22982.275,E2 -22982.275} C_VEL
LIN {X 0,Y 177.87,Z 443.013,A -85,B 0,C 180,E1 -22986.348,E2 -22986.348} C_VEL
LIN {X 0,Y 181.953,Z 437.608,A -85,B 0,C 180,E1 -22990.242,E2 -22990.242} C_VEL
LIN {X 0,Y 186.671,Z 430.621,A -85,B 0,C 180,E1 -22993.857,E2 -22993.857} C_VEL
LIN {X 0,Y 190.855,Z 423.529,A -85,B 0,C 180,E1 -22996.658,E2 -22996.658} C_VEL
LIN {X 0,Y 195.799,Z 414.233,A -85,B 0,C 180,E1 -22999.437,E2 -22999.437} C_VEL
LIN {X 0,Y 200.402,Z 404.369,A -85,B 0,C 180,E1 -23001.69,E2 -23001.69} C_VEL
LIN {X 0,Y 204.353,Z 394.282,A -85,B 0,C 180,E1 -23003.503,E2 -23003.503} C_VEL
LIN {X 0,Y 207.927,Z 383.183,A -85,B 0,C 180,E1 -23005.047,E2 -23005.047} C_VEL
LIN {X 0,Y 211.054,Z 370.785,A -85,B 0,C 180,E1 -23006.353,E2 -23006.353} C_VEL
LIN {X 0,Y 213.489,Z 357.706,A -85,B 0,C 180,E1 -23007.332,E2 -23007.332} C_VEL
LIN {X 0,Y 214.997,Z 344.989,A -85,B 0,C 180,E1 -23007.938,E2 -23007.938} C_VEL
LIN {X 0,Y 217.281,Z 311.543,A -85,B 0,C 180,E1 -23008.97,E2 -23008.97} C_VEL
LIN {X 0,Y 211.477,Z 300.824,A -85,B 0,C 180,E1 -23011.532,E2 -23011.532} C_VEL
LIN {X 0,Y 205.715,Z 291.519,A -85,B 0,C 180,E1 -23014.314,E2 -23014.314} C_VEL
LIN {X 0,Y 200.213,Z 283.379,A -85,B 0,C 180,E1 -23017.287,E2 -23017.287} C_VEL
LIN {X 0,Y 197.33,Z 279.429,A -85,B 0,C 180,E1 -23019,E2 -23019} C_VEL
LIN {X 0,Y 194.271,Z 275.282,A -85,B 0,C 180,E1 -23021,E2 -23021} C_VEL
LIN {X 0,Y 191.472,Z 271.648,A -85,B 0,C 180,E1 -23023.022,E2 -23023.022} C_VEL
LIN {X 0,Y 190.461,Z 270.34,A -85,B 0,C 180,E1 -23023.807,E2 -23023.807} C_VEL
LIN {X 0,Y 187.976,Z 267.421,A -85,B 0,C 180,E1 -23025.858,E2 -23025.858} C_VEL
LIN {X 0,Y 186.819,Z 265.527,A -85,B 0,C 180,E1 -23026.956,E2 -23026.956} C_VEL
LIN {X 0,Y 184.258,Z 263.284,A -85,B 0,C 180,E1 -23029.424,E2 -23029.424} C_VEL
LIN {X 0,Y 182.726,Z 260.225,A -85,B 0,C 180,E1 -23031.36,E2 -23031.36} C_VEL
LIN {X 0,Y 179.282,Z 257.693,A -85,B 0,C 180,E1 -23036.208,E2 -23036.208} C_VEL
LIN {X 0,Y 178.253,Z 255.156,A -85,B 0,C 180,E1 -23038.659,E2 -23038.659} C_VEL
LIN {X 0,Y 178.027,Z 254.13,A -85,B 0,C 180,E1 -23039.435,E2 -23039.435} C_VEL
LIN {X 0,Y 176.477,Z 253.863,A -85,B 0,C 180,E1 -23049.167,E2 -23049.167} C_VEL
LIN {X 0,Y 177.554,Z 254.353,A -85,B 0,C 180,E1 -23053.885,E2 -23053.885} C_VEL
LIN {X 0,Y 178.449,Z 256.901,A -85,B 0,C 180,E1 -23056.591,E2 -23056.591} C_VEL
LIN {X 0,Y 180.907,Z 259.499,A -85,B 0,C 180,E1 -23060.838,E2 -23060.838} C_VEL
LIN {X 0,Y 183.099,Z 261.836,A -85,B 0,C 180,E1 -23063.669,E2 -23063.669} C_VEL
LIN {X 0,Y 188.341,Z 269.255,A -85,B 0,C 180,E1 -23069.02,E2 -23069.02} C_VEL
LIN {X 0,Y 192.698,Z 275.778,A -85,B 0,C 180,E1 -23072.526,E2 -23072.526} C_VEL
LIN {X 0,Y 196.54,Z 281.91,A -85,B 0,C 180,E1 -23075.19,E2 -23075.19} C_VEL
LIN {X 0,Y 200.004,Z 287.728,A -85,B 0,C 180,E1 -23077.333,E2 -23077.333} C_VEL
LIN {X 0,Y 204.338,Z 295.288,A -85,B 0,C 180,E1 -23079.765,E2 -23079.765} C_VEL
LIN {X 0,Y 210.114,Z 306.88,A -85,B 0,C 180,E1 -23082.734,E2 -23082.734} C_VEL
LIN {X 0,Y 214.544,Z 317.312,A -85,B 0,C 180,E1 -23084.859,E2 -23084.859} C_VEL
LIN {X 0,Y 216.288,Z 322.173,A -85,B 0,C 180,E1 -23085.679,E2 -23085.679} C_VEL
LIN {X 0,Y 216.498,Z 325.475,A -85,B 0,C 180,E1 -23085.915,E2 -23085.915} C_VEL
LIN {X 0,Y 213.915,Z 361.389,A -85,B 0,C 180,E1 -23087.037,E2 -23087.037} C_VEL
LIN {X 0,Y 211.874,Z 374.972,A -85,B 0,C 180,E1 -23087.738,E2 -23087.738} C_VEL
LIN {X 0,Y 209.282,Z 386.607,A -85,B 0,C 180,E1 -23088.614,E2 -23088.614} C_VEL
LIN {X 0,Y 205.755,Z 398.621,A -85,B 0,C 180,E1 -23089.856,E2 -23089.856} C_VEL
LIN {X 0,Y 204.895,Z 401.136,A -85,B 0,C 180,E1 -23090.166,E2 -23090.166} C_VEL
LIN {X 0,Y 202.598,Z 406.229,A -85,B 0,C 180,E1 -23090.717,E2 -23090.717} C_VEL
LIN {X 0,Y 197.256,Z 414.23,A -85,B 0,C 180,E1 -23091.43,E2 -23091.43} C_VEL
LIN {X 0,Y 191.635,Z 421.745,A -85,B 0,C 180,E1 -23092.356,E2 -23092.356} C_VEL
LIN {X 0,Y 188.936,Z 426.072,A -85,B 0,C 180,E1 -23093.245,E2 -23093.245} C_VEL
LIN {X 0,Y 184.09,Z 434.857,A -85,B 0,C 180,E1 -23095.728,E2 -23095.728} C_VEL
LIN {X 0,Y 179.15,Z 442.889,A -85,B 0,C 180,E1 -23098.68,E2 -23098.68} C_VEL
LIN {X 0,Y 174.76,Z 449.473,A -85,B 0,C 180,E1 -23101.865,E2 -23101.865} C_VEL
LIN {X 0,Y 170.597,Z 455.293,A -85,B 0,C 180,E1 -23105.67,E2 -23105.67} C_VEL
LIN {X 0,Y 167.524,Z 459.186,A -85,B 0,C 180,E1 -23109.106,E2 -23109.106} C_VEL
LIN {X 0,Y 165.055,Z 462.085,A -85,B 0,C 180,E1 -23112.656,E2 -23112.656} C_VEL
LIN {X 0,Y 162.994,Z 464.497,A -85,B 0,C 180,E1 -23117.547,E2 -23117.547} C_VEL
LIN {X 0,Y 162.017,Z 465.377,A -85,B 0,C 180,E1 -23122.519,E2 -23122.519} C_VEL
LIN {X 0,Y 162.045,Z 464.654,A -85,B 0,C 180,E1 -23127.51,E2 -23127.51} C_VEL
LIN {X 0,Y 162.226,Z 463.708,A -85,B 0,C 180,E1 -23129.996,E2 -23129.996} C_VEL
LIN {X 0,Y 162.013,Z 461.334,A -85,B 0,C 180,E1 -23133.855,E2 -23133.855} C_VEL
LIN {X 0,Y 162.163,Z 458.13,A -85,B 0,C 180,E1 -23137.466,E2 -23137.466} C_VEL
LIN {X 0,Y 162.597,Z 453.715,A -85,B 0,C 180,E1 -23141.21,E2 -23141.21} C_VEL
LIN {X 0,Y 163.581,Z 448.07,A -85,B 0,C 180,E1 -23144.933,E2 -23144.933} C_VEL
LIN {X 0,Y 165.303,Z 441.014,A -85,B 0,C 180,E1 -23148.588,E2 -23148.588} C_VEL
LIN {X 0,Y 167.125,Z 433.779,A -85,B 0,C 180,E1 -23151.583,E2 -23151.583} C_VEL
LIN {X 0,Y 168.85,Z 427.015,A -85,B 0,C 180,E1 -23153.891,E2 -23153.891} C_VEL
LIN {X 0,Y 171.231,Z 417.706,A -85,B 0,C 180,E1 -23156.503,E2 -23156.503} C_VEL
LIN {X 0,Y 173.549,Z 407.703,A -85,B 0,C 180,E1 -23158.736,E2 -23158.736} C_VEL
LIN {X 0,Y 176.023,Z 396.873,A -85,B 0,C 180,E1 -23160.594,E2 -23160.594} C_VEL
LIN {X 0,Y 177.944,Z 386.028,A -85,B 0,C 180,E1 -23162.046,E2 -23162.046} C_VEL
LIN {X 0,Y 179.735,Z 373.584,A -85,B 0,C 180,E1 -23163.259,E2 -23163.259} C_VEL
LIN {X 0,Y 180.902,Z 361.074,A -85,B 0,C 180,E1 -23164.084,E2 -23164.084} C_VEL
LIN {X 0,Y 183.073,Z 315.381,A -85,B 0,C 180,E1 -23165.809,E2 -23165.809} C_VEL
LIN {X 0,Y 180.512,Z 288.399,A -85,B 0,C 180,E1 -23167.506,E2 -23167.506} C_VEL
LIN {X 0,Y 174.167,Z 271.332,A -85,B 0,C 180,E1 -23169.603,E2 -23169.603} C_VEL
LIN {X 0,Y 168.823,Z 259.668,A -85,B 0,C 180,E1 -23171.393,E2 -23171.393} C_VEL
LIN {X 0,Y 165.064,Z 251.895,A -85,B 0,C 180,E1 -23172.726,E2 -23172.726} C_VEL
LIN {X 0,Y 164.312,Z 249.016,A -85,B 0,C 180,E1 -23174.677,E2 -23174.677} C_VEL
LIN {X 0,Y 164.303,Z 249.015,A -85,B 0,C 180,E1 -23180.336,E2 -23180.336} C_VEL
LIN {X 0,Y 164.322,Z 249.014,A -85,B 0,C 180,E1 -23184.338,E2 -23184.338} C_VEL
LIN {X 0,Y 164.368,Z 249.009,A -85,B 0,C 180,E1 -23189.129,E2 -23189.129} C_VEL
LIN {X 0,Y 164.395,Z 249.005,A -85,B 0,C 180,E1 -23194.69,E2 -23194.69} C_VEL
LIN {X 0,Y 164.479,Z 248.993,A -85,B 0,C 180,E1 -23200.03,E2 -23200.03} C_VEL
LIN {X 0,Y 164.497,Z 248.995,A -85,B 0,C 180,E1 -23205.146,E2 -23205.146} C_VEL
LIN {X 0,Y 164.763,Z 248.957,A -85,B 0,C 180,E1 -23210.175,E2 -23210.175} C_VEL
LIN {X 0,Y 164.814,Z 248.954,A -85,B 0,C 180,E1 -23212.649,E2 -23212.649} C_VEL
LIN {X 0,Y 165.014,Z 248.887,A -85,B 0,C 180,E1 -23217.558,E2 -23217.558} C_VEL
LIN {X 0,Y 165.257,Z 248.845,A -85,B 0,C 180,E1 -23219.999,E2 -23219.999} C_VEL
LIN {X 0,Y 164.794,Z 248.957,A -85,B 0,C 180,E1 -23227.35,E2 -23227.35} C_VEL
LIN {X 0,Y 164.674,Z 248.958,A -85,B 0,C 180,E1 -23231.057,E2 -23231.057} C_VEL
LIN {X 0,Y 164.407,Z 249,A -85,B 0,C 180,E1 -23237.411,E2 -23237.411} C_VEL
LIN {X 0,Y 164.324,Z 249.015,A -85,B 0,C 180,E1 -23242.638,E2 -23242.638} C_VEL
LIN {X 0,Y 164.343,Z 249.002,A -85,B 0,C 180,E1 -23246.118,E2 -23246.118} C_VEL
LIN {X 0,Y 164.319,Z 248.967,A -85,B 0,C 180,E1 -23251.212,E2 -23251.212} C_VEL
LIN {X 0,Y 164.258,Z 249.023,A -85,B 0,C 180,E1 -23256.798,E2 -23256.798} C_VEL
LIN {X 0,Y 164.266,Z 249.01,A -85,B 0,C 180,E1 -23259.923,E2 -23259.923} C_VEL
LIN {X 0,Y 164.261,Z 248.989,A -85,B 0,C 180,E1 -23263.347,E2 -23263.347} C_VEL
LIN {X 0,Y 164.243,Z 249.022,A -85,B 0,C 180,E1 -23266.803,E2 -23266.803} C_VEL
LIN {X 0,Y 164.273,Z 249.012,A -85,B 0,C 180,E1 -23270.36,E2 -23270.36} C_VEL
LIN {X 0,Y 164.312,Z 249.019,A -85,B 0,C 180,E1 -23276.226,E2 -23276.226} C_VEL
LIN {X 0,Y 164.377,Z 248.994,A -85,B 0,C 180,E1 -23279.14,E2 -23279.14} C_VEL
LIN {X 0,Y 164.372,Z 249.102,A -85,B 0,C 180,E1 -23282.693,E2 -23282.693} C_VEL
LIN {X 0,Y 165.322,Z 251.772,A -85,B 0,C 180,E1 -23283.078,E2 -23283.078} C_VEL
LIN {X 0,Y 166.948,Z 254.151,A -85,B 0,C 180,E1 -23283.608,E2 -23283.608} C_VEL
LIN {X 0,Y 172.606,Z 264.05,A -85,B 0,C 180,E1 -23285.433,E2 -23285.433} C_VEL
LIN {X 0,Y 179.511,Z 277.575,A -85,B 0,C 180,E1 -23287.534,E2 -23287.534} C_VEL
LIN {X 0,Y 184.193,Z 288.371,A -85,B 0,C 180,E1 -23288.918,E2 -23288.918} C_VEL
LIN {X 0,Y 181.173,Z 347.314,A -85,B 0,C 180,E1 -23291.107,E2 -23291.107} C_VEL
LIN {X 0,Y 179.924,Z 361.177,A -85,B 0,C 180,E1 -23292.091,E2 -23292.091} C_VEL
LIN {X 0,Y 178.337,Z 373.498,A -85,B 0,C 180,E1 -23293.404,E2 -23293.404} C_VEL
LIN {X 0,Y 176.443,Z 384.57,A -85,B 0,C 180,E1 -23295,E2 -23295} C_VEL
LIN {X 0,Y 174.296,Z 394.846,A -85,B 0,C 180,E1 -23296.896,E2 -23296.896} C_VEL
LIN {X 0,Y 172.001,Z 405.124,A -85,B 0,C 180,E1 -23299.317,E2 -23299.317} C_VEL
LIN {X 0,Y 169.452,Z 415.062,A -85,B 0,C 180,E1 -23302.258,E2 -23302.258} C_VEL
LIN {X 0,Y 166.915,Z 424.296,A -85,B 0,C 180,E1 -23305.779,E2 -23305.779} C_VEL
LIN {X 0,Y 164.987,Z 431.718,A -85,B 0,C 180,E1 -23309.394,E2 -23309.394} C_VEL
LIN {X 0,Y 163.819,Z 436.746,A -85,B 0,C 180,E1 -23312.463,E2 -23312.463} C_VEL
LIN {X 0,Y 162.697,Z 442.023,A -85,B 0,C 180,E1 -23316.53,E2 -23316.53} C_VEL
LIN {X 0,Y 162.041,Z 445.419,A -85,B 0,C 180,E1 -23319.994,E2 -23319.994} C_VEL
LIN {X 0,Y 161.734,Z 447.383,A -85,B 0,C 180,E1 -23322.552,E2 -23322.552} C_VEL
LIN {X 0,Y 161.857,Z 449.752,A -85,B 0,C 180,E1 -23327.206,E2 -23327.206} C_VEL
LIN {X 0,Y 162.223,Z 450.575,A -85,B 0,C 180,E1 -23330.281,E2 -23330.281} C_VEL
LIN {X 0,Y 162.841,Z 450.805,A -85,B 0,C 180,E1 -23332.859,E2 -23332.859} C_VEL
LIN {X 0,Y 163.785,Z 450.537,A -85,B 0,C 180,E1 -23335.698,E2 -23335.698} C_VEL
LIN {X 0,Y 166.135,Z 448.914,A -85,B 0,C 180,E1 -23340.508,E2 -23340.508} C_VEL
LIN {X 0,Y 167.934,Z 447.24,A -85,B 0,C 180,E1 -23343.177,E2 -23343.177} C_VEL
LIN {X 0,Y 170.776,Z 444.215,A -85,B 0,C 180,E1 -23346.637,E2 -23346.637} C_VEL
LIN {X 0,Y 174.379,Z 439.895,A -85,B 0,C 180,E1 -23350.155,E2 -23350.155} C_VEL
LIN {X 0,Y 178.579,Z 434.282,A -85,B 0,C 180,E1 -23353.529,E2 -23353.529} C_VEL
LIN {X 0,Y 183.321,Z 427.18,A -85,B 0,C 180,E1 -23356.753,E2 -23356.753} C_VEL
LIN {X 0,Y 187.635,Z 419.823,A -85,B 0,C 180,E1 -23359.33,E2 -23359.33} C_VEL
LIN {X 0,Y 192.517,Z 410.452,A -85,B 0,C 180,E1 -23361.855,E2 -23361.855} C_VEL
LIN {X 0,Y 197.4,Z 399.605,A -85,B 0,C 180,E1 -23364.091,E2 -23364.091} C_VEL
LIN {X 0,Y 201.532,Z 388.474,A -85,B 0,C 180,E1 -23365.839,E2 -23365.839} C_VEL
LIN {X 0,Y 205.082,Z 376.217,A -85,B 0,C 180,E1 -23367.322,E2 -23367.322} C_VEL
LIN {X 0,Y 207.72,Z 364.641,A -85,B 0,C 180,E1 -23368.337,E2 -23368.337} C_VEL
LIN {X 0,Y 209.657,Z 352.436,A -85,B 0,C 180,E1 -23369.102,E2 -23369.102} C_VEL
LIN {X 0,Y 211.05,Z 336.706,A -85,B 0,C 180,E1 -23369.691,E2 -23369.691} C_VEL
LIN {X 0,Y 212.654,Z 314.551,A -85,B 0,C 180,E1 -23370.351,E2 -23370.351} C_VEL
LIN {X 0,Y 206.844,Z 303.775,A -85,B 0,C 180,E1 -23373.108,E2 -23373.108} C_VEL
LIN {X 0,Y 200.428,Z 293.484,A -85,B 0,C 180,E1 -23376.494,E2 -23376.494} C_VEL
LIN {X 0,Y 195.368,Z 286.049,A -85,B 0,C 180,E1 -23379.537,E2 -23379.537} C_VEL
LIN {X 0,Y 191.824,Z 281.267,A -85,B 0,C 180,E1 -23381.966,E2 -23381.966} C_VEL
LIN {X 0,Y 188.699,Z 276.954,A -85,B 0,C 180,E1 -23384.402,E2 -23384.402} C_VEL
LIN {X 0,Y 186.035,Z 273.658,A -85,B 0,C 180,E1 -23386.718,E2 -23386.718} C_VEL
LIN {X 0,Y 185.075,Z 272.158,A -85,B 0,C 180,E1 -23387.667,E2 -23387.667} C_VEL
LIN {X 0,Y 182.52,Z 269.607,A -85,B 0,C 180,E1 -23390.302,E2 -23390.302} C_VEL
LIN {X 0,Y 181.107,Z 266.853,A -85,B 0,C 180,E1 -23392.195,E2 -23392.195} C_VEL
LIN {X 0,Y 178.257,Z 264.688,A -85,B 0,C 180,E1 -23396.433,E2 -23396.433} C_VEL
LIN {X 0,Y 177.156,Z 262.143,A -85,B 0,C 180,E1 -23399.131,E2 -23399.131} C_VEL
LIN {X 0,Y 176.915,Z 261.101,A -85,B 0,C 180,E1 -23400.001,E2 -23400.001} C_VEL
LIN {X 0,Y 175.601,Z 260.911,A -85,B 0,C 180,E1 -23409.213,E2 -23409.213} C_VEL
LIN {X 0,Y 176.536,Z 261.439,A -85,B 0,C 180,E1 -23413.527,E2 -23413.527} C_VEL
LIN {X 0,Y 177.47,Z 263.986,A -85,B 0,C 180,E1 -23416.427,E2 -23416.427} C_VEL
LIN {X 0,Y 179.978,Z 266.559,A -85,B 0,C 180,E1 -23420.816,E2 -23420.816} C_VEL
LIN {X 0,Y 181.826,Z 268.887,A -85,B 0,C 180,E1 -23423.303,E2 -23423.303} C_VEL
LIN {X 0,Y 186.442,Z 275.605,A -85,B 0,C 180,E1 -23428.227,E2 -23428.227} C_VEL
LIN {X 0,Y 190.636,Z 282.159,A -85,B 0,C 180,E1 -23431.791,E2 -23431.791} C_VEL
LIN {X 0,Y 194.118,Z 287.958,A -85,B 0,C 180,E1 -23434.346,E2 -23434.346} C_VEL
LIN {X 0,Y 197.471,Z 293.813,A -85,B 0,C 180,E1 -23436.533,E2 -23436.533} C_VEL
LIN {X 0,Y 201.338,Z 300.857,A -85,B 0,C 180,E1 -23438.827,E2 -23438.827} C_VEL
LIN {X 0,Y 206.582,Z 311.677,A -85,B 0,C 180,E1 -23441.68,E2 -23441.68} C_VEL
LIN {X 0,Y 210.613,Z 321.509,A -85,B 0,C 180,E1 -23443.739,E2 -23443.739} C_VEL
LIN {X 0,Y 211.932,Z 325.342,A -85,B 0,C 180,E1 -23444.41,E2 -23444.41} C_VEL
LIN {X 0,Y 209.362,Z 360.749,A -85,B 0,C 180,E1 -23445.546,E2 -23445.546} C_VEL
LIN {X 0,Y 207.222,Z 374.672,A -85,B 0,C 180,E1 -23446.269,E2 -23446.269} C_VEL
LIN {X 0,Y 204.592,Z 385.99,A -85,B 0,C 180,E1 -23447.111,E2 -23447.111} C_VEL
LIN {X 0,Y 200.94,Z 398.083,A -85,B 0,C 180,E1 -23448.353,E2 -23448.353} C_VEL
LIN {X 0,Y 196.581,Z 409.591,A -85,B 0,C 180,E1 -23449.945,E2 -23449.945} C_VEL
LIN {X 0,Y 192.042,Z 419.961,A -85,B 0,C 180,E1 -23451.861,E2 -23451.861} C_VEL
LIN {X 0,Y 188.936,Z 426.072,A -85,B 0,C 180,E1 -23453.245,E2 -23453.245} C_VEL
LIN {X 0,Y 186.172,Z 430.284,A -85,B 0,C 180,E1 -23454.222,E2 -23454.222} C_VEL
LIN {X 0,Y 180.112,Z 436.734,A -85,B 0,C 180,E1 -23455.656,E2 -23455.656} C_VEL
LIN {X 0,Y 174.02,Z 442.513,A -85,B 0,C 180,E1 -23457.335,E2 -23457.335} C_VEL
LIN {X 0,Y 171.267,Z 445.713,A -85,B 0,C 180,E1 -23458.683,E2 -23458.683} C_VEL
LIN {X 0,Y 166.614,Z 452.149,A -85,B 0,C 180,E1 -23462.353,E2 -23462.353} C_VEL
LIN {X 0,Y 162.978,Z 456.68,A -85,B 0,C 180,E1 -23465.814,E2 -23465.814} C_VEL
LIN {X 0,Y 159.974,Z 460.159,A -85,B 0,C 180,E1 -23469.421,E2 -23469.421} C_VEL
LIN {X 0,Y 156.953,Z 463.273,A -85,B 0,C 180,E1 -23474.412,E2 -23474.412} C_VEL
LIN {X 0,Y 155.383,Z 464.853,A -85,B 0,C 180,E1 -23479.573,E2 -23479.573} C_VEL
LIN {X 0,Y 154.847,Z 464.826,A -85,B 0,C 180,E1 -23484.788,E2 -23484.788} C_VEL
LIN {X 0,Y 154.956,Z 464.241,A -85,B 0,C 180,E1 -23487.396,E2 -23487.396} C_VEL
LIN {X 0,Y 155.144,Z 463.262,A -85,B 0,C 180,E1 -23489.996,E2 -23489.996} C_VEL
LIN {X 0,Y 154.924,Z 461.111,A -85,B 0,C 180,E1 -23493.603,E2 -23493.603} C_VEL
LIN {X 0,Y 155.081,Z 457.536,A -85,B 0,C 180,E1 -23497.809,E2 -23497.809} C_VEL
LIN {X 0,Y 155.581,Z 453.04,A -85,B 0,C 180,E1 -23501.723,E2 -23501.723} C_VEL
LIN {X 0,Y 156.702,Z 447.311,A -85,B 0,C 180,E1 -23505.604,E2 -23505.604} C_VEL
LIN {X 0,Y 158.504,Z 440.101,A -85,B 0,C 180,E1 -23509.417,E2 -23509.417} C_VEL
LIN {X 0,Y 160.39,Z 432.734,A -85,B 0,C 180,E1 -23512.538,E2 -23512.538} C_VEL
LIN {X 0,Y 162.971,Z 423.834,A -85,B 0,C 180,E1 -23515.539,E2 -23515.539} C_VEL
LIN {X 0,Y 165.422,Z 414.002,A -85,B 0,C 180,E1 -23518.199,E2 -23518.199} C_VEL
LIN {X 0,Y 167.969,Z 403.244,A -85,B 0,C 180,E1 -23520.478,E2 -23520.478} C_VEL
LIN {X 0,Y 170.157,Z 393.186,A -85,B 0,C 180,E1 -23522.117,E2 -23522.117} C_VEL
LIN {X 0,Y 172.279,Z 381.294,A -85,B 0,C 180,E1 -23523.583,E2 -23523.583} C_VEL
LIN {X 0,Y 173.987,Z 368.34,A -85,B 0,C 180,E1 -23524.705,E2 -23524.705} C_VEL
LIN {X 0,Y 175.087,Z 354.975,A -85,B 0,C 180,E1 -23525.42,E2 -23525.42} C_VEL
LIN {X 0,Y 176.887,Z 316.073,A -85,B 0,C 180,E1 -23526.907,E2 -23526.907} C_VEL
LIN {X 0,Y 174.534,Z 290.499,A -85,B 0,C 180,E1 -23528.592,E2 -23528.592} C_VEL
LIN {X 0,Y 168.689,Z 274.541,A -85,B 0,C 180,E1 -23530.66,E2 -23530.66} C_VEL
LIN {X 0,Y 162.171,Z 260.292,A -85,B 0,C 180,E1 -23533.002,E2 -23533.002} C_VEL
LIN {X 0,Y 157.651,Z 251.404,A -85,B 0,C 180,E1 -23534.779,E2 -23534.779} C_VEL
LIN {X 0,Y 157.25,Z 249.898,A -85,B 0,C 180,E1 -23535.842,E2 -23535.842} C_VEL
LIN {X 0,Y 157.23,Z 249.898,A -85,B 0,C 180,E1 -23541.259,E2 -23541.259} C_VEL
LIN {X 0,Y 157.27,Z 249.893,A -85,B 0,C 180,E1 -23544.482,E2 -23544.482} C_VEL
LIN {X 0,Y 157.273,Z 249.891,A -85,B 0,C 180,E1 -23548.091,E2 -23548.091} C_VEL
LIN {X 0,Y 157.299,Z 249.891,A -85,B 0,C 180,E1 -23553.461,E2 -23553.461} C_VEL
LIN {X 0,Y 157.395,Z 249.877,A -85,B 0,C 180,E1 -23559.64,E2 -23559.64} C_VEL
LIN {X 0,Y 157.432,Z 249.874,A -85,B 0,C 180,E1 -23564.463,E2 -23564.463} C_VEL
LIN {X 0,Y 157.691,Z 249.834,A -85,B 0,C 180,E1 -23569.73,E2 -23569.73} C_VEL
LIN {X 0,Y 157.772,Z 249.831,A -85,B 0,C 180,E1 -23572.319,E2 -23572.319} C_VEL
LIN {X 0,Y 158.218,Z 249.719,A -85,B 0,C 180,E1 -23579.999,E2 -23579.999} C_VEL
LIN {X 0,Y 157.732,Z 249.835,A -85,B 0,C 180,E1 -23587.681,E2 -23587.681} C_VEL
LIN {X 0,Y 157.603,Z 249.838,A -85,B 0,C 180,E1 -23591.222,E2 -23591.222} C_VEL
LIN {X 0,Y 157.386,Z 249.88,A -85,B 0,C 180,E1 -23595.54,E2 -23595.54} C_VEL
LIN {X 0,Y 157.284,Z 249.883,A -85,B 0,C 180,E1 -23600.944,E2 -23600.944} C_VEL
LIN {X 0,Y 157.269,Z 249.878,A -85,B 0,C 180,E1 -23606.671,E2 -23606.671} C_VEL
LIN {X 0,Y 157.237,Z 249.856,A -85,B 0,C 180,E1 -23612.435,E2 -23612.435} C_VEL
LIN {X 0,Y 157.237,Z 249.895,A -85,B 0,C 180,E1 -23616.448,E2 -23616.448} C_VEL
LIN {X 0,Y 157.17,Z 249.872,A -85,B 0,C 180,E1 -23622.123,E2 -23622.123} C_VEL
LIN {X 0,Y 157.173,Z 249.907,A -85,B 0,C 180,E1 -23627.888,E2 -23627.888} C_VEL
LIN {X 0,Y 157.244,Z 249.878,A -85,B 0,C 180,E1 -23633.561,E2 -23633.561} C_VEL
LIN {X 0,Y 157.28,Z 249.883,A -85,B 0,C 180,E1 -23638.102,E2 -23638.102} C_VEL
LIN {X 0,Y 157.278,Z 249.881,A -85,B 0,C 180,E1 -23640.799,E2 -23640.799} C_VEL
LIN {X 0,Y 158.221,Z 252.669,A -85,B 0,C 180,E1 -23641.25,E2 -23641.25} C_VEL
LIN {X 0,Y 159.914,Z 255.023,A -85,B 0,C 180,E1 -23641.85,E2 -23641.85} C_VEL
LIN {X 0,Y 166.107,Z 265.458,A -85,B 0,C 180,E1 -23644.001,E2 -23644.001} C_VEL
LIN {X 0,Y 173.556,Z 279.936,A -85,B 0,C 180,E1 -23646.426,E2 -23646.426} C_VEL
LIN {X 0,Y 178.006,Z 290.289,A -85,B 0,C 180,E1 -23647.835,E2 -23647.835} C_VEL
LIN {X 0,Y 174.964,Z 347.298,A -85,B 0,C 180,E1 -23650.004,E2 -23650.004} C_VEL
LIN {X 0,Y 173.732,Z 360.565,A -85,B 0,C 180,E1 -23650.951,E2 -23650.951} C_VEL
LIN {X 0,Y 172.055,Z 373.288,A -85,B 0,C 180,E1 -23652.32,E2 -23652.32} C_VEL
LIN {X 0,Y 169.886,Z 385.301,A -85,B 0,C 180,E1 -23654.099,E2 -23654.099} C_VEL
LIN {X 0,Y 167.397,Z 396.786,A -85,B 0,C 180,E1 -23656.346,E2 -23656.346} C_VEL
LIN {X 0,Y 165.007,Z 406.688,A -85,B 0,C 180,E1 -23658.826,E2 -23658.826} C_VEL
LIN {X 0,Y 162.365,Z 416.437,A -85,B 0,C 180,E1 -23661.918,E2 -23661.918} C_VEL
LIN {X 0,Y 159.791,Z 425.477,A -85,B 0,C 180,E1 -23665.59,E2 -23665.59} C_VEL
LIN {X 0,Y 157.838,Z 432.747,A -85,B 0,C 180,E1 -23669.367,E2 -23669.367} C_VEL
LIN {X 0,Y 156.625,Z 437.651,A -85,B 0,C 180,E1 -23672.576,E2 -23672.576} C_VEL
LIN {X 0,Y 155.596,Z 442.376,A -85,B 0,C 180,E1 -23676.442,E2 -23676.442} C_VEL
LIN {X 0,Y 154.865,Z 446.096,A -85,B 0,C 180,E1 -23680.462,E2 -23680.462} C_VEL
LIN {X 0,Y 154.608,Z 447.969,A -85,B 0,C 180,E1 -23683.141,E2 -23683.141} C_VEL
LIN {X 0,Y 154.781,Z 450.068,A -85,B 0,C 180,E1 -23687.539,E2 -23687.539} C_VEL
LIN {X 0,Y 155.302,Z 450.983,A -85,B 0,C 180,E1 -23691.228,E2 -23691.228} C_VEL
LIN {X 0,Y 156.912,Z 450.881,A -85,B 0,C 180,E1 -23696.392,E2 -23696.392} C_VEL
LIN {X 0,Y 158.219,Z 450.168,A -85,B 0,C 180,E1 -23699.252,E2 -23699.252} C_VEL
LIN {X 0,Y 161.357,Z 447.625,A -85,B 0,C 180,E1 -23704.153,E2 -23704.153} C_VEL
LIN {X 0,Y 164.83,Z 444.147,A -85,B 0,C 180,E1 -23708.19,E2 -23708.19} C_VEL
LIN {X 0,Y 168.73,Z 439.704,A -85,B 0,C 180,E1 -23711.794,E2 -23711.794} C_VEL
LIN {X 0,Y 173.236,Z 433.96,A -85,B 0,C 180,E1 -23715.232,E2 -23715.232} C_VEL
LIN {X 0,Y 178.267,Z 426.655,A -85,B 0,C 180,E1 -23718.509,E2 -23718.509} C_VEL
LIN {X 0,Y 182.875,Z 419.12,A -85,B 0,C 180,E1 -23721.097,E2 -23721.097} C_VEL
LIN {X 0,Y 187.903,Z 409.846,A -85,B 0,C 180,E1 -23723.555,E2 -23723.555} C_VEL
LIN {X 0,Y 192.608,Z 399.682,A -85,B 0,C 180,E1 -23725.643,E2 -23725.643} C_VEL
LIN {X 0,Y 196.927,Z 388.316,A -85,B 0,C 180,E1 -23727.428,E2 -23727.428} C_VEL
LIN {X 0,Y 200.584,Z 376.111,A -85,B 0,C 180,E1 -23728.894,E2 -23728.894} C_VEL
LIN {X 0,Y 203.565,Z 363.229,A -85,B 0,C 180,E1 -23729.983,E2 -23729.983} C_VEL
LIN {X 0,Y 205.546,Z 350.107,A -85,B 0,C 180,E1 -23730.747,E2 -23730.747} C_VEL
LIN {X 0,Y 207.441,Z 327.653,A -85,B 0,C 180,E1 -23731.476,E2 -23731.476} C_VEL
LIN {X 0,Y 208.157,Z 317.589,A -85,B 0,C 180,E1 -23731.792,E2 -23731.792} C_VEL
LIN {X 0,Y 202.873,Z 307.772,A -85,B 0,C 180,E1 -23734.478,E2 -23734.478} C_VEL
LIN {X 0,Y 197.007,Z 298.221,A -85,B 0,C 180,E1 -23737.796,E2 -23737.796} C_VEL
LIN {X 0,Y 192.742,Z 291.79,A -85,B 0,C 180,E1 -23740.548,E2 -23740.548} C_VEL
LIN {X 0,Y 189.706,Z 287.501,A -85,B 0,C 180,E1 -23742.761,E2 -23742.761} C_VEL
LIN {X 0,Y 186.797,Z 283.406,A -85,B 0,C 180,E1 -23745.14,E2 -23745.14} C_VEL
LIN {X 0,Y 184.068,Z 279.762,A -85,B 0,C 180,E1 -23747.669,E2 -23747.669} C_VEL
LIN {X 0,Y 183.362,Z 278.772,A -85,B 0,C 180,E1 -23748.392,E2 -23748.392} C_VEL
LIN {X 0,Y 180.828,Z 275.921,A -85,B 0,C 180,E1 -23751.198,E2 -23751.198} C_VEL
LIN {X 0,Y 179.778,Z 273.74,A -85,B 0,C 180,E1 -23752.702,E2 -23752.702} C_VEL
LIN {X 0,Y 177.077,Z 271.485,A -85,B 0,C 180,E1 -23756.979,E2 -23756.979} C_VEL
LIN {X 0,Y 176.004,Z 268.771,A -85,B 0,C 180,E1 -23759.876,E2 -23759.876} C_VEL
LIN {X 0,Y 175.795,Z 268.108,A -85,B 0,C 180,E1 -23760.631,E2 -23760.631} C_VEL
LIN {X 0,Y 175.123,Z 268.106,A -85,B 0,C 180,E1 -23771.576,E2 -23771.576} C_VEL
LIN {X 0,Y 175.537,Z 268.439,A -85,B 0,C 180,E1 -23773.163,E2 -23773.163} C_VEL
LIN {X 0,Y 176.602,Z 271.219,A -85,B 0,C 180,E1 -23776.51,E2 -23776.51} C_VEL
LIN {X 0,Y 179.425,Z 274.234,A -85,B 0,C 180,E1 -23781.364,E2 -23781.364} C_VEL
LIN {X 0,Y 180.679,Z 276.085,A -85,B 0,C 180,E1 -23783.081,E2 -23783.081} C_VEL
LIN {X 0,Y 184.711,Z 282.189,A -85,B 0,C 180,E1 -23787.551,E2 -23787.551} C_VEL
LIN {X 0,Y 188.61,Z 288.52,A -85,B 0,C 180,E1 -23791.035,E2 -23791.035} C_VEL
LIN {X 0,Y 191.83,Z 294.147,A -85,B 0,C 180,E1 -23793.536,E2 -23793.536} C_VEL
LIN {X 0,Y 194.85,Z 299.641,A -85,B 0,C 180,E1 -23795.629,E2 -23795.629} C_VEL
LIN {X 0,Y 198.849,Z 307.385,A -85,B 0,C 180,E1 -23798.138,E2 -23798.138} C_VEL
LIN {X 0,Y 203.64,Z 317.722,A -85,B 0,C 180,E1 -23800.878,E2 -23800.878} C_VEL
LIN {X 0,Y 207.355,Z 327.431,A -85,B 0,C 180,E1 -23802.897,E2 -23802.897} C_VEL
LIN {X 0,Y 207.422,Z 329.327,A -85,B 0,C 180,E1 -23803.031,E2 -23803.031} C_VEL
LIN {X 0,Y 204.873,Z 361.13,A -85,B 0,C 180,E1 -23804.036,E2 -23804.036} C_VEL
LIN {X 0,Y 202.673,Z 374.677,A -85,B 0,C 180,E1 -23804.744,E2 -23804.744} C_VEL
LIN {X 0,Y 199.793,Z 386.566,A -85,B 0,C 180,E1 -23805.643,E2 -23805.643} C_VEL
LIN {X 0,Y 195.736,Z 399.179,A -85,B 0,C 180,E1 -23806.984,E2 -23806.984} C_VEL
LIN {X 0,Y 191.234,Z 410.419,A -85,B 0,C 180,E1 -23808.584,E2 -23808.584} C_VEL
LIN {X 0,Y 186.544,Z 420.566,A -85,B 0,C 180,E1 -23810.523,E2 -23810.523} C_VEL
LIN {X 0,Y 182.059,Z 428.909,A -85,B 0,C 180,E1 -23812.555,E2 -23812.555} C_VEL
LIN {X 0,Y 176.545,Z 437.988,A -85,B 0,C 180,E1 -23815.439,E2 -23815.439} C_VEL
LIN {X 0,Y 171.267,Z 445.713,A -85,B 0,C 180,E1 -23818.683,E2 -23818.683} C_VEL
LIN {X 0,Y 168.563,Z 448.725,A -85,B 0,C 180,E1 -23820.138,E2 -23820.138} C_VEL
LIN {X 0,Y 162.653,Z 453.115,A -85,B 0,C 180,E1 -23822.444,E2 -23822.444} C_VEL
LIN {X 0,Y 156.906,Z 456.833,A -85,B 0,C 180,E1 -23825.029,E2 -23825.029} C_VEL
LIN {X 0,Y 154.53,Z 458.704,A -85,B 0,C 180,E1 -23826.895,E2 -23826.895} C_VEL
LIN {X 0,Y 151.544,Z 461.741,A -85,B 0,C 180,E1 -23831.054,E2 -23831.054} C_VEL
LIN {X 0,Y 149.078,Z 464.011,A -85,B 0,C 180,E1 -23836.363,E2 -23836.363} C_VEL
LIN {X 0,Y 148.368,Z 464.549,A -85,B 0,C 180,E1 -23839.074,E2 -23839.074} C_VEL
LIN {X 0,Y 147.776,Z 464.446,A -85,B 0,C 180,E1 -23844.538,E2 -23844.538} C_VEL
LIN {X 0,Y 147.886,Z 463.828,A -85,B 0,C 180,E1 -23847.272,E2 -23847.272} C_VEL
LIN {X 0,Y 148.063,Z 462.802,A -85,B 0,C 180,E1 -23849.995,E2 -23849.995} C_VEL
LIN {X 0,Y 147.84,Z 460.879,A -85,B 0,C 180,E1 -23853.333,E2 -23853.333} C_VEL
LIN {X 0,Y 148.016,Z 456.936,A -85,B 0,C 180,E1 -23858.184,E2 -23858.184} C_VEL
LIN {X 0,Y 148.588,Z 452.356,A -85,B 0,C 180,E1 -23862.283,E2 -23862.283} C_VEL
LIN {X 0,Y 150.144,Z 445.386,A -85,B 0,C 180,E1 -23867.004,E2 -23867.004} C_VEL
LIN {X 0,Y 152.153,Z 437.803,A -85,B 0,C 180,E1 -23870.969,E2 -23870.969} C_VEL
LIN {X 0,Y 154.274,Z 430.039,A -85,B 0,C 180,E1 -23874.197,E2 -23874.197} C_VEL
LIN {X 0,Y 157.076,Z 420.616,A -85,B 0,C 180,E1 -23877.29,E2 -23877.29} C_VEL
LIN {X 0,Y 159.846,Z 410.083,A -85,B 0,C 180,E1 -23880,E2 -23880} C_VEL
LIN {X 0,Y 162.284,Z 399.984,A -85,B 0,C 180,E1 -23882.031,E2 -23882.031} C_VEL
LIN {X 0,Y 164.767,Z 388.158,A -85,B 0,C 180,E1 -23883.852,E2 -23883.852} C_VEL
LIN {X 0,Y 166.783,Z 375.964,A -85,B 0,C 180,E1 -23885.215,E2 -23885.215} C_VEL
LIN {X 0,Y 168.335,Z 362.29,A -85,B 0,C 180,E1 -23886.234,E2 -23886.234} C_VEL
LIN {X 0,Y 169.798,Z 337.551,A -85,B 0,C 180,E1 -23887.262,E2 -23887.262} C_VEL
LIN {X 0,Y 170.73,Z 316.673,A -85,B 0,C 180,E1 -23888.098,E2 -23888.098} C_VEL
LIN {X 0,Y 168.672,Z 292.658,A -85,B 0,C 180,E1 -23889.74,E2 -23889.74} C_VEL
LIN {X 0,Y 162.74,Z 276.571,A -85,B 0,C 180,E1 -23891.974,E2 -23891.974} C_VEL
LIN {X 0,Y 157.024,Z 264.115,A -85,B 0,C 180,E1 -23894.172,E2 -23894.172} C_VEL
LIN {X 0,Y 152.253,Z 254.969,A -85,B 0,C 180,E1 -23896.111,E2 -23896.111} C_VEL
LIN {X 0,Y 150.565,Z 252.26,A -85,B 0,C 180,E1 -23896.808,E2 -23896.808} C_VEL
LIN {X 0,Y 150.234,Z 250.894,A -85,B 0,C 180,E1 -23897.101,E2 -23897.101} C_VEL
LIN {X 0,Y 150.2,Z 250.772,A -85,B 0,C 180,E1 -23902.683,E2 -23902.683} C_VEL
LIN {X 0,Y 150.197,Z 250.769,A -85,B 0,C 180,E1 -23907.362,E2 -23907.362} C_VEL
LIN {X 0,Y 150.223,Z 250.77,A -85,B 0,C 180,E1 -23912.714,E2 -23912.714} C_VEL
LIN {X 0,Y 150.345,Z 250.757,A -85,B 0,C 180,E1 -23919.188,E2 -23919.188} C_VEL
LIN {X 0,Y 150.343,Z 250.755,A -85,B 0,C 180,E1 -23923.71,E2 -23923.71} C_VEL
LIN {X 0,Y 150.616,Z 250.712,A -85,B 0,C 180,E1 -23929.242,E2 -23929.242} C_VEL
LIN {X 0,Y 150.707,Z 250.711,A -85,B 0,C 180,E1 -23931.957,E2 -23931.957} C_VEL
LIN {X 0,Y 151.178,Z 250.594,A -85,B 0,C 180,E1 -23939.999,E2 -23939.999} C_VEL
LIN {X 0,Y 150.67,Z 250.715,A -85,B 0,C 180,E1 -23948.043,E2 -23948.043} C_VEL
LIN {X 0,Y 150.546,Z 250.717,A -85,B 0,C 180,E1 -23951.426,E2 -23951.426} C_VEL
LIN {X 0,Y 150.291,Z 250.764,A -85,B 0,C 180,E1 -23956.294,E2 -23956.294} C_VEL
LIN {X 0,Y 150.258,Z 250.756,A -85,B 0,C 180,E1 -23960.725,E2 -23960.725} C_VEL
LIN {X 0,Y 150.204,Z 250.748,A -85,B 0,C 180,E1 -23967.272,E2 -23967.272} C_VEL
LIN {X 0,Y 150.178,Z 250.735,A -85,B 0,C 180,E1 -23972.627,E2 -23972.627} C_VEL
LIN {X 0,Y 150.149,Z 250.78,A -85,B 0,C 180,E1 -23977.479,E2 -23977.479} C_VEL
LIN {X 0,Y 150.112,Z 250.754,A -85,B 0,C 180,E1 -23981.501,E2 -23981.501} C_VEL
LIN {X 0,Y 150.108,Z 250.766,A -85,B 0,C 180,E1 -23985.4,E2 -23985.4} C_VEL
LIN {X 0,Y 150.121,Z 250.784,A -85,B 0,C 180,E1 -23989.059,E2 -23989.059} C_VEL
LIN {X 0,Y 150.161,Z 250.756,A -85,B 0,C 180,E1 -23992.716,E2 -23992.716} C_VEL
LIN {X 0,Y 150.219,Z 250.758,A -85,B 0,C 180,E1 -23998.688,E2 -23998.688} C_VEL
LIN {X 0,Y 151.274,Z 253.706,A -85,B 0,C 180,E1 -23999.252,E2 -23999.252} C_VEL
LIN {X 0,Y 153.009,Z 256.07,A -85,B 0,C 180,E1 -23999.932,E2 -23999.932} C_VEL
LIN {X 0,Y 159.597,Z 266.836,A -85,B 0,C 180,E1 -24002.428,E2 -24002.428} C_VEL
LIN {X 0,Y 167.381,Z 281.845,A -85,B 0,C 180,E1 -24005.153,E2 -24005.153} C_VEL
LIN {X 0,Y 171.907,Z 292.046,A -85,B 0,C 180,E1 -24006.671,E2 -24006.671} C_VEL
LIN {X 0,Y 168.774,Z 348.163,A -85,B 0,C 180,E1 -24008.877,E2 -24008.877} C_VEL
LIN {X 0,Y 167.398,Z 361.749,A -85,B 0,C 180,E1 -24009.891,E2 -24009.891} C_VEL
LIN {X 0,Y 165.672,Z 374.149,A -85,B 0,C 180,E1 -24011.294,E2 -24011.294} C_VEL
LIN {X 0,Y 163.377,Z 386.031,A -85,B 0,C 180,E1 -24013.126,E2 -24013.126} C_VEL
LIN {X 0,Y 160.8,Z 397.436,A -85,B 0,C 180,E1 -24015.451,E2 -24015.451} C_VEL
LIN {X 0,Y 158.335,Z 407.208,A -85,B 0,C 180,E1 -24018.002,E2 -24018.002} C_VEL
LIN {X 0,Y 155.805,Z 416.143,A -85,B 0,C 180,E1 -24020.922,E2 -24020.922} C_VEL
LIN {X 0,Y 153.051,Z 425.291,A -85,B 0,C 180,E1 -24024.736,E2 -24024.736} C_VEL
LIN {X 0,Y 150.962,Z 432.654,A -85,B 0,C 180,E1 -24028.671,E2 -24028.671} C_VEL
LIN {X 0,Y 149.442,Z 438.551,A -85,B 0,C 180,E1 -24032.7,E2 -24032.7} C_VEL
LIN {X 0,Y 148.494,Z 442.721,A -85,B 0,C 180,E1 -24036.34,E2 -24036.34} C_VEL
LIN {X 0,Y 147.684,Z 446.761,A -85,B 0,C 180,E1 -24040.977,E2 -24040.977} C_VEL
LIN {X 0,Y 147.51,Z 448.537,A -85,B 0,C 180,E1 -24043.785,E2 -24043.785} C_VEL
LIN {X 0,Y 147.718,Z 450.386,A -85,B 0,C 180,E1 -24047.912,E2 -24047.912} C_VEL
LIN {X 0,Y 148.431,Z 451.352,A -85,B 0,C 180,E1 -24052.262,E2 -24052.262} C_VEL
LIN {X 0,Y 150.086,Z 451.221,A -85,B 0,C 180,E1 -24057.166,E2 -24057.166} C_VEL
LIN {X 0,Y 151.749,Z 450.352,A -85,B 0,C 180,E1 -24060.629,E2 -24060.629} C_VEL
LIN {X 0,Y 154.827,Z 448.015,A -85,B 0,C 180,E1 -24065.209,E2 -24065.209} C_VEL
LIN {X 0,Y 159.027,Z 444.088,A -85,B 0,C 180,E1 -24069.854,E2 -24069.854} C_VEL
LIN {X 0,Y 163.249,Z 439.53,A -85,B 0,C 180,E1 -24073.537,E2 -24073.537} C_VEL
LIN {X 0,Y 168.053,Z 433.634,A -85,B 0,C 180,E1 -24077.042,E2 -24077.042} C_VEL
LIN {X 0,Y 173.366,Z 426.131,A -85,B 0,C 180,E1 -24080.375,E2 -24080.375} C_VEL
LIN {X 0,Y 178.281,Z 418.426,A -85,B 0,C 180,E1 -24082.965,E2 -24082.965} C_VEL
LIN {X 0,Y 183.336,Z 409.418,A -85,B 0,C 180,E1 -24085.311,E2 -24085.311} C_VEL
LIN {X 0,Y 187.945,Z 399.746,A -85,B 0,C 180,E1 -24087.283,E2 -24087.283} C_VEL
LIN {X 0,Y 192.608,Z 387.873,A -85,B 0,C 180,E1 -24089.121,E2 -24089.121} C_VEL
LIN {X 0,Y 196.262,Z 376.016,A -85,B 0,C 180,E1 -24090.528,E2 -24090.528} C_VEL
LIN {X 0,Y 199.254,Z 363.354,A -85,B 0,C 180,E1 -24091.59,E2 -24091.59} C_VEL
LIN {X 0,Y 201.289,Z 350.293,A -85,B 0,C 180,E1 -24092.347,E2 -24092.347} C_VEL
LIN {X 0,Y 203.519,Z 324.901,A -85,B 0,C 180,E1 -24093.146,E2 -24093.146} C_VEL
LIN {X 0,Y 203.79,Z 320.797,A -85,B 0,C 180,E1 -24093.289,E2 -24093.289} C_VEL
LIN {X 0,Y 199.117,Z 311.966,A -85,B 0,C 180,E1 -24095.845,E2 -24095.845} C_VEL
LIN {X 0,Y 193.015,Z 301.796,A -85,B 0,C 180,E1 -24099.597,E2 -24099.597} C_VEL
LIN {X 0,Y 189.472,Z 296.561,A -85,B 0,C 180,E1 -24102.112,E2 -24102.112} C_VEL
LIN {X 0,Y 187.577,Z 293.735,A -85,B 0,C 180,E1 -24103.602,E2 -24103.602} C_VEL
LIN {X 0,Y 184.745,Z 289.647,A -85,B 0,C 180,E1 -24106.055,E2 -24106.055} C_VEL
LIN {X 0,Y 181.685,Z 285.336,A -85,B 0,C 180,E1 -24109.131,E2 -24109.131} C_VEL
LIN {X 0,Y 179.282,Z 282.389,A -85,B 0,C 180,E1 -24111.973,E2 -24111.973} C_VEL
LIN {X 0,Y 178.27,Z 280.479,A -85,B 0,C 180,E1 -24113.493,E2 -24113.493} C_VEL
LIN {X 0,Y 175.832,Z 278.172,A -85,B 0,C 180,E1 -24117.71,E2 -24117.71} C_VEL
LIN {X 0,Y 174.75,Z 275.124,A -85,B 0,C 180,E1 -24121.108,E2 -24121.108} C_VEL
LIN {X 0,Y 174.258,Z 275.156,A -85,B 0,C 180,E1 -24131.635,E2 -24131.635} C_VEL
LIN {X 0,Y 174.542,Z 275.454,A -85,B 0,C 180,E1 -24132.795,E2 -24132.795} C_VEL
LIN {X 0,Y 175.692,Z 278.396,A -85,B 0,C 180,E1 -24136.5,E2 -24136.5} C_VEL
LIN {X 0,Y 178.217,Z 281.134,A -85,B 0,C 180,E1 -24140.97,E2 -24140.97} C_VEL
LIN {X 0,Y 179.861,Z 283.871,A -85,B 0,C 180,E1 -24143.287,E2 -24143.287} C_VEL
LIN {X 0,Y 183.008,Z 288.755,A -85,B 0,C 180,E1 -24146.862,E2 -24146.862} C_VEL
LIN {X 0,Y 186.576,Z 294.808,A -85,B 0,C 180,E1 -24150.229,E2 -24150.229} C_VEL
LIN {X 0,Y 189.323,Z 299.817,A -85,B 0,C 180,E1 -24152.498,E2 -24152.498} C_VEL
LIN {X 0,Y 192.508,Z 305.939,A -85,B 0,C 180,E1 -24154.863,E2 -24154.863} C_VEL
LIN {X 0,Y 196.147,Z 313.331,A -85,B 0,C 180,E1 -24157.273,E2 -24157.273} C_VEL
LIN {X 0,Y 200.426,Z 323.051,A -85,B 0,C 180,E1 -24159.874,E2 -24159.874} C_VEL
LIN {X 0,Y 203.107,Z 330.287,A -85,B 0,C 180,E1 -24161.436,E2 -24161.436} C_VEL
LIN {X 0,Y 200.6,Z 360.884,A -85,B 0,C 180,E1 -24162.427,E2 -24162.427} C_VEL
LIN {X 0,Y 198.35,Z 374.335,A -85,B 0,C 180,E1 -24163.131,E2 -24163.131} C_VEL
LIN {X 0,Y 195.425,Z 386.048,A -85,B 0,C 180,E1 -24164.007,E2 -24164.007} C_VEL
LIN {X 0,Y 191.821,Z 397.139,A -85,B 0,C 180,E1 -24165.147,E2 -24165.147} C_VEL
LIN {X 0,Y 187.171,Z 408.685,A -85,B 0,C 180,E1 -24166.744,E2 -24166.744} C_VEL
LIN {X 0,Y 182.191,Z 419.096,A -85,B 0,C 180,E1 -24168.654,E2 -24168.654} C_VEL
LIN {X 0,Y 177.471,Z 427.63,A -85,B 0,C 180,E1 -24170.682,E2 -24170.682} C_VEL
LIN {X 0,Y 172.568,Z 435.522,A -85,B 0,C 180,E1 -24173.078,E2 -24173.078} C_VEL
LIN {X 0,Y 167.202,Z 443.281,A -85,B 0,C 180,E1 -24176.154,E2 -24176.154} C_VEL
LIN {X 0,Y 163.158,Z 448.593,A -85,B 0,C 180,E1 -24178.874,E2 -24178.874} C_VEL
LIN {X 0,Y 159.088,Z 453.681,A -85,B 0,C 180,E1 -24182.257,E2 -24182.257} C_VEL
LIN {X 0,Y 155.337,Z 457.877,A -85,B 0,C 180,E1 -24185.969,E2 -24185.969} C_VEL
LIN {X 0,Y 154.53,Z 458.704,A -85,B 0,C 180,E1 -24186.895,E2 -24186.895} C_VEL
LIN {X 0,Y 152.309,Z 460.359,A -85,B 0,C 180,E1 -24188.848,E2 -24188.848} C_VEL
LIN {X 0,Y 147.351,Z 462.415,A -85,B 0,C 180,E1 -24192.038,E2 -24192.038} C_VEL
LIN {X 0,Y 142.903,Z 463.713,A -85,B 0,C 180,E1 -24195.496,E2 -24195.496} C_VEL
LIN {X 0,Y 141.544,Z 464.115,A -85,B 0,C 180,E1 -24197.8,E2 -24197.8} C_VEL
LIN {X 0,Y 140.889,Z 464.339,A -85,B 0,C 180,E1 -24201.389,E2 -24201.389} C_VEL
LIN {X 0,Y 140.807,Z 463.414,A -85,B 0,C 180,E1 -24207.134,E2 -24207.134} C_VEL
LIN {X 0,Y 140.985,Z 462.321,A -85,B 0,C 180,E1 -24209.995,E2 -24209.995} C_VEL
LIN {X 0,Y 140.779,Z 460.561,A -85,B 0,C 180,E1 -24213.178,E2 -24213.178} C_VEL
LIN {X 0,Y 140.838,Z 457.592,A -85,B 0,C 180,E1 -24217.161,E2 -24217.161} C_VEL
LIN {X 0,Y 141.342,Z 453.317,A -85,B 0,C 180,E1 -24221.466,E2 -24221.466} C_VEL
LIN {X 0,Y 142.704,Z 446.797,A -85,B 0,C 180,E1 -24226.443,E2 -24226.443} C_VEL
LIN {X 0,Y 144.681,Z 439.632,A -85,B 0,C 180,E1 -24230.613,E2 -24230.613} C_VEL
LIN {X 0,Y 146.615,Z 432.839,A -85,B 0,C 180,E1 -24233.792,E2 -24233.792} C_VEL
LIN {X 0,Y 149.59,Z 423.45,A -85,B 0,C 180,E1 -24237.254,E2 -24237.254} C_VEL
LIN {X 0,Y 152.289,Z 413.671,A -85,B 0,C 180,E1 -24240.116,E2 -24240.116} C_VEL
LIN {X 0,Y 155.062,Z 402.983,A -85,B 0,C 180,E1 -24242.554,E2 -24242.554} C_VEL
LIN {X 0,Y 157.433,Z 393.018,A -85,B 0,C 180,E1 -24244.296,E2 -24244.296} C_VEL
LIN {X 0,Y 159.708,Z 381.335,A -85,B 0,C 180,E1 -24245.852,E2 -24245.852} C_VEL
LIN {X 0,Y 161.646,Z 367.872,A -85,B 0,C 180,E1 -24247.094,E2 -24247.094} C_VEL
LIN {X 0,Y 162.844,Z 354.653,A -85,B 0,C 180,E1 -24247.844,E2 -24247.844} C_VEL
LIN {X 0,Y 164.722,Z 317.584,A -85,B 0,C 180,E1 -24249.346,E2 -24249.346} C_VEL
LIN {X 0,Y 162.821,Z 294.685,A -85,B 0,C 180,E1 -24250.985,E2 -24250.985} C_VEL
LIN {X 0,Y 157.065,Z 279.001,A -85,B 0,C 180,E1 -24253.307,E2 -24253.307} C_VEL
LIN {X 0,Y 151.77,Z 267.466,A -85,B 0,C 180,E1 -24255.497,E2 -24255.497} C_VEL
LIN {X 0,Y 147.746,Z 259.663,A -85,B 0,C 180,E1 -24257.255,E2 -24257.255} C_VEL
LIN {X 0,Y 145.527,Z 256.153,A -85,B 0,C 180,E1 -24258.235,E2 -24258.235} C_VEL
LIN {X 0,Y 143.72,Z 253.769,A -85,B 0,C 180,E1 -24259.035,E2 -24259.035} C_VEL
LIN {X 0,Y 143.089,Z 251.659,A -85,B 0,C 180,E1 -24259.487,E2 -24259.487} C_VEL
LIN {X 0,Y 143.093,Z 251.656,A -85,B 0,C 180,E1 -24263.886,E2 -24263.886} C_VEL
LIN {X 0,Y 143.164,Z 251.645,A -85,B 0,C 180,E1 -24267.316,E2 -24267.316} C_VEL
LIN {X 0,Y 143.14,Z 251.654,A -85,B 0,C 180,E1 -24273.775,E2 -24273.775} C_VEL
LIN {X 0,Y 143.299,Z 251.631,A -85,B 0,C 180,E1 -24279.92,E2 -24279.92} C_VEL
LIN {X 0,Y 143.341,Z 251.628,A -85,B 0,C 180,E1 -24285.808,E2 -24285.808} C_VEL
LIN {X 0,Y 143.551,Z 251.59,A -85,B 0,C 180,E1 -24288.706,E2 -24288.706} C_VEL
LIN {X 0,Y 143.627,Z 251.594,A -85,B 0,C 180,E1 -24291.558,E2 -24291.558} C_VEL
LIN {X 0,Y 144.136,Z 251.469,A -85,B 0,C 180,E1 -24299.999,E2 -24299.999} C_VEL
LIN {X 0,Y 143.592,Z 251.596,A -85,B 0,C 180,E1 -24308.443,E2 -24308.443} C_VEL
LIN {X 0,Y 143.471,Z 251.597,A -85,B 0,C 180,E1 -24311.611,E2 -24311.611} C_VEL
LIN {X 0,Y 143.23,Z 251.639,A -85,B 0,C 180,E1 -24317.121,E2 -24317.121} C_VEL
LIN {X 0,Y 143.197,Z 251.638,A -85,B 0,C 180,E1 -24321.198,E2 -24321.198} C_VEL
LIN {X 0,Y 143.15,Z 251.616,A -85,B 0,C 180,E1 -24327.927,E2 -24327.927} C_VEL
LIN {X 0,Y 143.111,Z 251.623,A -85,B 0,C 180,E1 -24333.417,E2 -24333.417} C_VEL
LIN {X 0,Y 143.032,Z 251.654,A -85,B 0,C 180,E1 -24339.699,E2 -24339.699} C_VEL
LIN {X 0,Y 143.014,Z 251.631,A -85,B 0,C 180,E1 -24343.47,E2 -24343.47} C_VEL
LIN {X 0,Y 143.021,Z 251.669,A -85,B 0,C 180,E1 -24347.483,E2 -24347.483} C_VEL
LIN {X 0,Y 143.056,Z 251.641,A -85,B 0,C 180,E1 -24351.816,E2 -24351.816} C_VEL
LIN {X 0,Y 143.14,Z 251.757,A -85,B 0,C 180,E1 -24356.362,E2 -24356.362} C_VEL
LIN {X 0,Y 144.152,Z 254.521,A -85,B 0,C 180,E1 -24356.916,E2 -24356.916} C_VEL
LIN {X 0,Y 146.094,Z 256.965,A -85,B 0,C 180,E1 -24357.758,E2 -24357.758} C_VEL
LIN {X 0,Y 153.772,Z 269.421,A -85,B 0,C 180,E1 -24360.957,E2 -24360.957} C_VEL
LIN {X 0,Y 159.063,Z 279.251,A -85,B 0,C 180,E1 -24362.979,E2 -24362.979} C_VEL
LIN {X 0,Y 165.064,Z 292.115,A -85,B 0,C 180,E1 -24365.151,E2 -24365.151} C_VEL
LIN {X 0,Y 165.802,Z 293.887,A -85,B 0,C 180,E1 -24365.413,E2 -24365.413} C_VEL
LIN {X 0,Y 162.668,Z 348.487,A -85,B 0,C 180,E1 -24367.628,E2 -24367.628} C_VEL
LIN {X 0,Y 161.221,Z 362.159,A -85,B 0,C 180,E1 -24368.678,E2 -24368.678} C_VEL
LIN {X 0,Y 159.346,Z 374.967,A -85,B 0,C 180,E1 -24370.187,E2 -24370.187} C_VEL
LIN {X 0,Y 156.938,Z 386.748,A -85,B 0,C 180,E1 -24372.075,E2 -24372.075} C_VEL
LIN {X 0,Y 154.246,Z 398.085,A -85,B 0,C 180,E1 -24374.48,E2 -24374.48} C_VEL
LIN {X 0,Y 151.605,Z 407.972,A -85,B 0,C 180,E1 -24377.176,E2 -24377.176} C_VEL
LIN {X 0,Y 148.75,Z 417.499,A -85,B 0,C 180,E1 -24380.487,E2 -24380.487} C_VEL
LIN {X 0,Y 145.948,Z 426.471,A -85,B 0,C 180,E1 -24384.479,E2 -24384.479} C_VEL
LIN {X 0,Y 143.825,Z 433.667,A -85,B 0,C 180,E1 -24388.605,E2 -24388.605} C_VEL
LIN {X 0,Y 142.262,Z 439.403,A -85,B 0,C 180,E1 -24392.836,E2 -24392.836} C_VEL
LIN {X 0,Y 141.216,Z 443.829,A -85,B 0,C 180,E1 -24397.034,E2 -24397.034} C_VEL
LIN {X 0,Y 140.536,Z 447.385,A -85,B 0,C 180,E1 -24401.543,E2 -24401.543} C_VEL
LIN {X 0,Y 140.412,Z 449.106,A -85,B 0,C 180,E1 -24404.497,E2 -24404.497} C_VEL
LIN {X 0,Y 140.666,Z 450.705,A -85,B 0,C 180,E1 -24408.329,E2 -24408.329} C_VEL
LIN {X 0,Y 141.592,Z 451.718,A -85,B 0,C 180,E1 -24413.399,E2 -24413.399} C_VEL
LIN {X 0,Y 143.246,Z 451.57,A -85,B 0,C 180,E1 -24417.98,E2 -24417.98} C_VEL
LIN {X 0,Y 145.384,Z 450.515,A -85,B 0,C 180,E1 -24422.126,E2 -24422.126} C_VEL
LIN {X 0,Y 148.393,Z 448.395,A -85,B 0,C 180,E1 -24426.379,E2 -24426.379} C_VEL
LIN {X 0,Y 151.992,Z 445.303,A -85,B 0,C 180,E1 -24430.344,E2 -24430.344} C_VEL
LIN {X 0,Y 156.599,Z 440.735,A -85,B 0,C 180,E1 -24434.382,E2 -24434.382} C_VEL
LIN {X 0,Y 162.168,Z 434.401,A -85,B 0,C 180,E1 -24438.381,E2 -24438.381} C_VEL
LIN {X 0,Y 167.625,Z 427.149,A -85,B 0,C 180,E1 -24441.732,E2 -24441.732} C_VEL
LIN {X 0,Y 173.755,Z 417.965,A -85,B 0,C 180,E1 -24444.854,E2 -24444.854} C_VEL
LIN {X 0,Y 178.887,Z 409.131,A -85,B 0,C 180,E1 -24447.115,E2 -24447.115} C_VEL
LIN {X 0,Y 184.037,Z 398.463,A -85,B 0,C 180,E1 -24449.229,E2 -24449.229} C_VEL
LIN {X 0,Y 188.542,Z 387.127,A -85,B 0,C 180,E1 -24450.944,E2 -24450.944} C_VEL
LIN {X 0,Y 192.103,Z 375.918,A -85,B 0,C 180,E1 -24452.236,E2 -24452.236} C_VEL
LIN {X 0,Y 195.167,Z 363.154,A -85,B 0,C 180,E1 -24453.289,E2 -24453.289} C_VEL
LIN {X 0,Y 197.233,Z 350.199,A -85,B 0,C 180,E1 -24454.028,E2 -24454.028} C_VEL
LIN {X 0,Y 199.553,Z 323.927,A -85,B 0,C 180,E1 -24454.861,E2 -24454.861} C_VEL
LIN {X 0,Y 195.161,Z 315.713,A -85,B 0,C 180,E1 -24457.452,E2 -24457.452} C_VEL
LIN {X 0,Y 190.437,Z 307.516,A -85,B 0,C 180,E1 -24460.602,E2 -24460.602} C_VEL
LIN {X 0,Y 185.75,Z 300.266,A -85,B 0,C 180,E1 -24464.247,E2 -24464.247} C_VEL
LIN {X 0,Y 182.65,Z 295.74,A -85,B 0,C 180,E1 -24467.077,E2 -24467.077} C_VEL
LIN {X 0,Y 180.035,Z 291.913,A -85,B 0,C 180,E1 -24469.883,E2 -24469.883} C_VEL
LIN {X 0,Y 177.682,Z 288.699,A -85,B 0,C 180,E1 -24472.9,E2 -24472.9} C_VEL
LIN {X 0,Y 176.999,Z 287.318,A -85,B 0,C 180,E1 -24474.018,E2 -24474.018} C_VEL
LIN {X 0,Y 174.707,Z 285.001,A -85,B 0,C 180,E1 -24478.229,E2 -24478.229} C_VEL
LIN {X 0,Y 173.771,Z 282.145,A -85,B 0,C 180,E1 -24481.415,E2 -24481.415} C_VEL
LIN {X 0,Y 173.475,Z 282.226,A -85,B 0,C 180,E1 -24492.021,E2 -24492.021} C_VEL
LIN {X 0,Y 175.163,Z 286.087,A -85,B 0,C 180,E1 -24497.325,E2 -24497.325} C_VEL
LIN {X 0,Y 176.96,Z 287.945,A -85,B 0,C 180,E1 -24500.468,E2 -24500.468} C_VEL
LIN {X 0,Y 178.975,Z 291.592,A -85,B 0,C 180,E1 -24503.409,E2 -24503.409} C_VEL
LIN {X 0,Y 181.211,Z 295.077,A -85,B 0,C 180,E1 -24506.024,E2 -24506.024} C_VEL
LIN {X 0,Y 184.493,Z 300.979,A -85,B 0,C 180,E1 -24509.332,E2 -24509.332} C_VEL
LIN {X 0,Y 186.925,Z 305.623,A -85,B 0,C 180,E1 -24511.476,E2 -24511.476} C_VEL
LIN {X 0,Y 190.811,Z 313.369,A -85,B 0,C 180,E1 -24514.51,E2 -24514.51} C_VEL
LIN {X 0,Y 195.351,Z 323.555,A -85,B 0,C 180,E1 -24517.61,E2 -24517.61} C_VEL
LIN {X 0,Y 198.67,Z 332.267,A -85,B 0,C 180,E1 -24519.714,E2 -24519.714} C_VEL
LIN {X 0,Y 198.909,Z 332.95,A -85,B 0,C 180,E1 -24519.862,E2 -24519.862} C_VEL
LIN {X 0,Y 196.561,Z 360.262,A -85,B 0,C 180,E1 -24520.741,E2 -24520.741} C_VEL
LIN {X 0,Y 194.242,Z 373.754,A -85,B 0,C 180,E1 -24521.433,E2 -24521.433} C_VEL
LIN {X 0,Y 191.113,Z 385.905,A -85,B 0,C 180,E1 -24522.331,E2 -24522.331} C_VEL
LIN {X 0,Y 186.882,Z 398.243,A -85,B 0,C 180,E1 -24523.621,E2 -24523.621} C_VEL
LIN {X 0,Y 182.103,Z 409.526,A -85,B 0,C 180,E1 -24525.224,E2 -24525.224} C_VEL
LIN {X 0,Y 176.957,Z 419.73,A -85,B 0,C 180,E1 -24527.145,E2 -24527.145} C_VEL
LIN {X 0,Y 172.068,Z 428.102,A -85,B 0,C 180,E1 -24529.193,E2 -24529.193} C_VEL
LIN {X 0,Y 166.004,Z 437.21,A -85,B 0,C 180,E1 -24532.128,E2 -24532.128} C_VEL
LIN {X 0,Y 160.466,Z 444.578,A -85,B 0,C 180,E1 -24535.292,E2 -24535.292} C_VEL
LIN {X 0,Y 155.594,Z 450.521,A -85,B 0,C 180,E1 -24538.703,E2 -24538.703} C_VEL
LIN {X 0,Y 151.398,Z 455.249,A -85,B 0,C 180,E1 -24542.339,E2 -24542.339} C_VEL
LIN {X 0,Y 147.716,Z 458.9,A -85,B 0,C 180,E1 -24546.143,E2 -24546.143} C_VEL
LIN {X 0,Y 144.816,Z 461.573,A -85,B 0,C 180,E1 -24550.137,E2 -24550.137} C_VEL
LIN {X 0,Y 143.256,Z 462.86,A -85,B 0,C 180,E1 -24552.878,E2 -24552.878} C_VEL
LIN {X 0,Y 141.544,Z 464.115,A -85,B 0,C 180,E1 -24557.8,E2 -24557.8} C_VEL
LIN {X 0,Y 140.476,Z 464.339,A -85,B 0,C 180,E1 -24560.158,E2 -24560.158} C_VEL
LIN {X 0,Y 138.757,Z 464.227,A -85,B 0,C 180,E1 -24562.488,E2 -24562.488} C_VEL
LIN {X 0,Y 135.078,Z 463.04,A -85,B 0,C 180,E1 -24567.23,E2 -24567.23} C_VEL
LIN {X 0,Y 133.83,Z 461.552,A -85,B 0,C 180,E1 -24570.527,E2 -24570.527} C_VEL
LIN {X 0,Y 133.668,Z 459.282,A -85,B 0,C 180,E1 -24574.518,E2 -24574.518} C_VEL
LIN {X 0,Y 133.936,Z 455.682,A -85,B 0,C 180,E1 -24579.051,E2 -24579.051} C_VEL
LIN {X 0,Y 134.659,Z 450.919,A -85,B 0,C 180,E1 -24583.577,E2 -24583.577} C_VEL
LIN {X 0,Y 136.197,Z 444.877,A -85,B 0,C 180,E1 -24588.029,E2 -24588.029} C_VEL
LIN {X 0,Y 138.43,Z 437.324,A -85,B 0,C 180,E1 -24592.374,E2 -24592.374} C_VEL
LIN {X 0,Y 140.892,Z 429.269,A -85,B 0,C 180,E1 -24596.026,E2 -24596.026} C_VEL
LIN {X 0,Y 143.831,Z 420.225,A -85,B 0,C 180,E1 -24599.242,E2 -24599.242} C_VEL
LIN {X 0,Y 146.876,Z 409.745,A -85,B 0,C 180,E1 -24602.154,E2 -24602.154} C_VEL
LIN {X 0,Y 149.548,Z 399.717,A -85,B 0,C 180,E1 -24604.319,E2 -24604.319} C_VEL
LIN {X 0,Y 152.002,Z 388.978,A -85,B 0,C 180,E1 -24606.113,E2 -24606.113} C_VEL
LIN {X 0,Y 154.436,Z 376.026,A -85,B 0,C 180,E1 -24607.689,E2 -24607.689} C_VEL
LIN {X 0,Y 156.093,Z 362.868,A -85,B 0,C 180,E1 -24608.755,E2 -24608.755} C_VEL
LIN {X 0,Y 157.313,Z 344.801,A -85,B 0,C 180,E1 -24609.601,E2 -24609.601} C_VEL
LIN {X 0,Y 158.722,Z 317.861,A -85,B 0,C 180,E1 -24610.726,E2 -24610.726} C_VEL
LIN {X 0,Y 157.111,Z 296.971,A -85,B 0,C 180,E1 -24612.282,E2 -24612.282} C_VEL
LIN {X 0,Y 151.935,Z 282.642,A -85,B 0,C 180,E1 -24614.534,E2 -24614.534} C_VEL
LIN {X 0,Y 146.543,Z 270.65,A -85,B 0,C 180,E1 -24616.947,E2 -24616.947} C_VEL
LIN {X 0,Y 143.307,Z 264.348,A -85,B 0,C 180,E1 -24618.469,E2 -24618.469} C_VEL
LIN {X 0,Y 141.032,Z 260.883,A -85,B 0,C 180,E1 -24619.536,E2 -24619.536} C_VEL
LIN {X 0,Y 138.609,Z 257.183,A -85,B 0,C 180,E1 -24620.734,E2 -24620.734} C_VEL
LIN {X 0,Y 136.813,Z 254.981,A -85,B 0,C 180,E1 -24621.621,E2 -24621.621} C_VEL
LIN {X 0,Y 136.049,Z 252.537,A -85,B 0,C 180,E1 -24622.16,E2 -24622.16} C_VEL
LIN {X 0,Y 136.072,Z 252.533,A -85,B 0,C 180,E1 -24625.713,E2 -24625.713} C_VEL
LIN {X 0,Y 136.126,Z 252.524,A -85,B 0,C 180,E1 -24632.311,E2 -24632.311} C_VEL
LIN {X 0,Y 136.239,Z 252.515,A -85,B 0,C 180,E1 -24638.831,E2 -24638.831} C_VEL
LIN {X 0,Y 136.25,Z 252.514,A -85,B 0,C 180,E1 -24645.053,E2 -24645.053} C_VEL
LIN {X 0,Y 136.475,Z 252.471,A -85,B 0,C 180,E1 -24648.112,E2 -24648.112} C_VEL
LIN {X 0,Y 136.554,Z 252.473,A -85,B 0,C 180,E1 -24651.117,E2 -24651.117} C_VEL
LIN {X 0,Y 137.093,Z 252.344,A -85,B 0,C 180,E1 -24659.999,E2 -24659.999} C_VEL
LIN {X 0,Y 136.518,Z 252.474,A -85,B 0,C 180,E1 -24668.883,E2 -24668.883} C_VEL
LIN {X 0,Y 136.389,Z 252.479,A -85,B 0,C 180,E1 -24671.894,E2 -24671.894} C_VEL
LIN {X 0,Y 136.141,Z 252.515,A -85,B 0,C 180,E1 -24678.042,E2 -24678.042} C_VEL
LIN {X 0,Y 136.123,Z 252.523,A -85,B 0,C 180,E1 -24681.696,E2 -24681.696} C_VEL
LIN {X 0,Y 136.061,Z 252.488,A -85,B 0,C 180,E1 -24688.606,E2 -24688.606} C_VEL
LIN {X 0,Y 136.017,Z 252.522,A -85,B 0,C 180,E1 -24694.635,E2 -24694.635} C_VEL
LIN {X 0,Y 136.004,Z 252.533,A -85,B 0,C 180,E1 -24699.199,E2 -24699.199} C_VEL
LIN {X 0,Y 135.959,Z 252.509,A -85,B 0,C 180,E1 -24703.653,E2 -24703.653} C_VEL
LIN {X 0,Y 135.966,Z 252.548,A -85,B 0,C 180,E1 -24707.793,E2 -24707.793} C_VEL
LIN {X 0,Y 136.028,Z 252.517,A -85,B 0,C 180,E1 -24713.535,E2 -24713.535} C_VEL
LIN {X 0,Y 137.137,Z 255.535,A -85,B 0,C 180,E1 -24714.291,E2 -24714.291} C_VEL
LIN {X 0,Y 139.192,Z 257.91,A -85,B 0,C 180,E1 -24715.29,E2 -24715.29} C_VEL
LIN {X 0,Y 141.39,Z 261.233,A -85,B 0,C 180,E1 -24716.364,E2 -24716.364} C_VEL
LIN {X 0,Y 148.648,Z 273,A -85,B 0,C 180,E1 -24719.622,E2 -24719.622} C_VEL
LIN {X 0,Y 154.031,Z 283.169,A -85,B 0,C 180,E1 -24721.838,E2 -24721.838} C_VEL
LIN {X 0,Y 159.854,Z 295.901,A -85,B 0,C 180,E1 -24724.099,E2 -24724.099} C_VEL
LIN {X 0,Y 156.644,Z 348.619,A -85,B 0,C 180,E1 -24726.279,E2 -24726.279} C_VEL
LIN {X 0,Y 155.138,Z 362.349,A -85,B 0,C 180,E1 -24727.359,E2 -24727.359} C_VEL
LIN {X 0,Y 153.257,Z 374.697,A -85,B 0,C 180,E1 -24728.837,E2 -24728.837} C_VEL
LIN {X 0,Y 150.953,Z 385.804,A -85,B 0,C 180,E1 -24730.633,E2 -24730.633} C_VEL
LIN {X 0,Y 148.377,Z 396.095,A -85,B 0,C 180,E1 -24732.787,E2 -24732.787} C_VEL
LIN {X 0,Y 145.521,Z 406.713,A -85,B 0,C 180,E1 -24735.676,E2 -24735.676} C_VEL
LIN {X 0,Y 142.81,Z 415.432,A -85,B 0,C 180,E1 -24738.653,E2 -24738.653} C_VEL
LIN {X 0,Y 140.203,Z 423.458,A -85,B 0,C 180,E1 -24742.082,E2 -24742.082} C_VEL
LIN {X 0,Y 137.683,Z 431.301,A -85,B 0,C 180,E1 -24746.347,E2 -24746.347} C_VEL
LIN {X 0,Y 136.082,Z 436.65,A -85,B 0,C 180,E1 -24750.005,E2 -24750.005} C_VEL
LIN {X 0,Y 134.702,Z 441.845,A -85,B 0,C 180,E1 -24754.493,E2 -24754.493} C_VEL
LIN {X 0,Y 133.763,Z 445.899,A -85,B 0,C 180,E1 -24759.073,E2 -24759.073} C_VEL
LIN {X 0,Y 133.396,Z 447.996,A -85,B 0,C 180,E1 -24762.17,E2 -24762.17} C_VEL
LIN {X 0,Y 133.344,Z 449.667,A -85,B 0,C 180,E1 -24765.284,E2 -24765.284} C_VEL
LIN {X 0,Y 133.605,Z 451.015,A -85,B 0,C 180,E1 -24768.767,E2 -24768.767} C_VEL
LIN {X 0,Y 134.811,Z 452.083,A -85,B 0,C 180,E1 -24774.652,E2 -24774.652} C_VEL
LIN {X 0,Y 136.441,Z 451.919,A -85,B 0,C 180,E1 -24778.879,E2 -24778.879} C_VEL
LIN {X 0,Y 139.113,Z 450.679,A -85,B 0,C 180,E1 -24783.763,E2 -24783.763} C_VEL
LIN {X 0,Y 142.009,Z 448.784,A -85,B 0,C 180,E1 -24787.644,E2 -24787.644} C_VEL
LIN {X 0,Y 146.372,Z 445.251,A -85,B 0,C 180,E1 -24792.239,E2 -24792.239} C_VEL
LIN {X 0,Y 151.038,Z 440.883,A -85,B 0,C 180,E1 -24796.115,E2 -24796.115} C_VEL
LIN {X 0,Y 156.359,Z 435.142,A -85,B 0,C 180,E1 -24799.829,E2 -24799.829} C_VEL
LIN {X 0,Y 162.182,Z 427.898,A -85,B 0,C 180,E1 -24803.291,E2 -24803.291} C_VEL
LIN {X 0,Y 168.61,Z 418.731,A -85,B 0,C 180,E1 -24806.474,E2 -24806.474} C_VEL
LIN {X 0,Y 174.384,Z 409.243,A -85,B 0,C 180,E1 -24808.915,E2 -24808.915} C_VEL
LIN {X 0,Y 179.746,Z 398.515,A -85,B 0,C 180,E1 -24811.026,E2 -24811.026} C_VEL
LIN {X 0,Y 184.307,Z 387.41,A -85,B 0,C 180,E1 -24812.699,E2 -24812.699} C_VEL
LIN {X 0,Y 188.318,Z 375.047,A -85,B 0,C 180,E1 -24814.094,E2 -24814.094} C_VEL
LIN {X 0,Y 191.482,Z 361.763,A -85,B 0,C 180,E1 -24815.147,E2 -24815.147} C_VEL
LIN {X 0,Y 193.439,Z 349.481,A -85,B 0,C 180,E1 -24815.804,E2 -24815.804} C_VEL
LIN {X 0,Y 195.411,Z 327.089,A -85,B 0,C 180,E1 -24816.528,E2 -24816.528} C_VEL
LIN {X 0,Y 191.302,Z 319.342,A -85,B 0,C 180,E1 -24819.167,E2 -24819.167} C_VEL
LIN {X 0,Y 186.823,Z 311.432,A -85,B 0,C 180,E1 -24822.486,E2 -24822.486} C_VEL
LIN {X 0,Y 183.482,Z 306.2,A -85,B 0,C 180,E1 -24825.312,E2 -24825.312} C_VEL
LIN {X 0,Y 180.987,Z 302.323,A -85,B 0,C 180,E1 -24827.74,E2 -24827.74} C_VEL
LIN {X 0,Y 178.534,Z 298.573,A -85,B 0,C 180,E1 -24830.513,E2 -24830.513} C_VEL
LIN {X 0,Y 176.309,Z 295.376,A -85,B 0,C 180,E1 -24833.555,E2 -24833.555} C_VEL
LIN {X 0,Y 175.652,Z 294.113,A -85,B 0,C 180,E1 -24834.683,E2 -24834.683} C_VEL
LIN {X 0,Y 173.491,Z 291.613,A -85,B 0,C 180,E1 -24839.046,E2 -24839.046} C_VEL
LIN {X 0,Y 172.797,Z 289.166,A -85,B 0,C 180,E1 -24841.726,E2 -24841.726} C_VEL
LIN {X 0,Y 172.529,Z 289.254,A -85,B 0,C 180,E1 -24851.753,E2 -24851.753} C_VEL
LIN {X 0,Y 174.001,Z 292.892,A -85,B 0,C 180,E1 -24856.764,E2 -24856.764} C_VEL
LIN {X 0,Y 175.892,Z 294.986,A -85,B 0,C 180,E1 -24860.239,E2 -24860.239} C_VEL
LIN {X 0,Y 179.533,Z 301.587,A -85,B 0,C 180,E1 -24865.274,E2 -24865.274} C_VEL
LIN {X 0,Y 182.675,Z 307.518,A -85,B 0,C 180,E1 -24868.626,E2 -24868.626} C_VEL
LIN {X 0,Y 185.341,Z 312.974,A -85,B 0,C 180,E1 -24871.093,E2 -24871.093} C_VEL
LIN {X 0,Y 189.389,Z 321.67,A -85,B 0,C 180,E1 -24874.368,E2 -24874.368} C_VEL
LIN {X 0,Y 193.491,Z 331.738,A -85,B 0,C 180,E1 -24877.29,E2 -24877.29} C_VEL
LIN {X 0,Y 194.833,Z 335.49,A -85,B 0,C 180,E1 -24878.198,E2 -24878.198} C_VEL
LIN {X 0,Y 192.587,Z 360.372,A -85,B 0,C 180,E1 -24879.013,E2 -24879.013} C_VEL
LIN {X 0,Y 190.219,Z 373.61,A -85,B 0,C 180,E1 -24879.69,E2 -24879.69} C_VEL
LIN {X 0,Y 187.049,Z 385.514,A -85,B 0,C 180,E1 -24880.558,E2 -24880.558} C_VEL
LIN {X 0,Y 182.73,Z 397.772,A -85,B 0,C 180,E1 -24881.825,E2 -24881.825} C_VEL
LIN {X 0,Y 177.771,Z 409.083,A -85,B 0,C 180,E1 -24883.411,E2 -24883.411} C_VEL
LIN {X 0,Y 172.424,Z 419.31,A -85,B 0,C 180,E1 -24885.323,E2 -24885.323} C_VEL
LIN {X 0,Y 166.773,Z 428.524,A -85,B 0,C 180,E1 -24887.603,E2 -24887.603} C_VEL
LIN {X 0,Y 160.459,Z 437.498,A -85,B 0,C 180,E1 -24890.572,E2 -24890.572} C_VEL
LIN {X 0,Y 154.675,Z 444.758,A -85,B 0,C 180,E1 -24893.793,E2 -24893.793} C_VEL
LIN {X 0,Y 149.56,Z 450.605,A -85,B 0,C 180,E1 -24897.287,E2 -24897.287} C_VEL
LIN {X 0,Y 145.113,Z 455.245,A -85,B 0,C 180,E1 -24901.03,E2 -24901.03} C_VEL
LIN {X 0,Y 141.231,Z 458.813,A -85,B 0,C 180,E1 -24904.974,E2 -24904.974} C_VEL
LIN {X 0,Y 138.132,Z 461.41,A -85,B 0,C 180,E1 -24909.133,E2 -24909.133} C_VEL
LIN {X 0,Y 136.454,Z 462.657,A -85,B 0,C 180,E1 -24911.996,E2 -24911.996} C_VEL
LIN {X 0,Y 134.411,Z 463.926,A -85,B 0,C 180,E1 -24917.923,E2 -24917.923} C_VEL
LIN {X 0,Y 133.627,Z 463.683,A -85,B 0,C 180,E1 -24923.957,E2 -24923.957} C_VEL
LIN {X 0,Y 133.72,Z 462.98,A -85,B 0,C 180,E1 -24926.982,E2 -24926.982} C_VEL
LIN {X 0,Y 133.83,Z 461.552,A -85,B 0,C 180,E1 -24930.527,E2 -24930.527} C_VEL
LIN {X 0,Y 132.996,Z 460.239,A -85,B 0,C 180,E1 -24932.964,E2 -24932.964} C_VEL
LIN {X 0,Y 130.154,Z 457.351,A -85,B 0,C 180,E1 -24936.919,E2 -24936.919} C_VEL
LIN {X 0,Y 128.028,Z 454.56,A -85,B 0,C 180,E1 -24940.12,E2 -24940.12} C_VEL
LIN {X 0,Y 127.396,Z 452.13,A -85,B 0,C 180,E1 -24942.552,E2 -24942.552} C_VEL
LIN {X 0,Y 127.485,Z 451.255,A -85,B 0,C 180,E1 -24943.355,E2 -24943.355} C_VEL
LIN {X 0,Y 129.092,Z 445.169,A -85,B 0,C 180,E1 -24948.235,E2 -24948.235} C_VEL
LIN {X 0,Y 131.358,Z 437.743,A -85,B 0,C 180,E1 -24952.815,E2 -24952.815} C_VEL
LIN {X 0,Y 133.143,Z 432.104,A -85,B 0,C 180,E1 -24955.659,E2 -24955.659} C_VEL
LIN {X 0,Y 136.376,Z 422.996,A -85,B 0,C 180,E1 -24959.304,E2 -24959.304} C_VEL
LIN {X 0,Y 139.356,Z 413.255,A -85,B 0,C 180,E1 -24962.391,E2 -24962.391} C_VEL
LIN {X 0,Y 142.385,Z 402.61,A -85,B 0,C 180,E1 -24965.006,E2 -24965.006} C_VEL
LIN {X 0,Y 144.973,Z 392.712,A -85,B 0,C 180,E1 -24966.854,E2 -24966.854} C_VEL
LIN {X 0,Y 147.431,Z 381.161,A -85,B 0,C 180,E1 -24968.502,E2 -24968.502} C_VEL
LIN {X 0,Y 149.532,Z 367.909,A -85,B 0,C 180,E1 -24969.809,E2 -24969.809} C_VEL
LIN {X 0,Y 150.824,Z 355.11,A -85,B 0,C 180,E1 -24970.599,E2 -24970.599} C_VEL
LIN {X 0,Y 152.855,Z 318.469,A -85,B 0,C 180,E1 -24972.182,E2 -24972.182} C_VEL
LIN {X 0,Y 151.466,Z 299.287,A -85,B 0,C 180,E1 -24973.681,E2 -24973.681} C_VEL
LIN {X 0,Y 146.692,Z 285.819,A -85,B 0,C 180,E1 -24975.934,E2 -24975.934} C_VEL
LIN {X 0,Y 140.83,Z 272.548,A -85,B 0,C 180,E1 -24978.805,E2 -24978.805} C_VEL
LIN {X 0,Y 137.652,Z 266.75,A -85,B 0,C 180,E1 -24980.424,E2 -24980.424} C_VEL
LIN {X 0,Y 134.275,Z 262.026,A -85,B 0,C 180,E1 -24982.166,E2 -24982.166} C_VEL
LIN {X 0,Y 132.275,Z 258.817,A -85,B 0,C 180,E1 -24983.291,E2 -24983.291} C_VEL
LIN {X 0,Y 129.753,Z 255.826,A -85,B 0,C 180,E1 -24984.709,E2 -24984.709} C_VEL
LIN {X 0,Y 129.033,Z 253.411,A -85,B 0,C 180,E1 -24985.307,E2 -24985.307} C_VEL
LIN {X 0,Y 128.998,Z 253.41,A -85,B 0,C 180,E1 -24990.636,E2 -24990.636} C_VEL
LIN {X 0,Y 129.014,Z 253.413,A -85,B 0,C 180,E1 -24994.163,E2 -24994.163} C_VEL
LIN {X 0,Y 129.097,Z 253.402,A -85,B 0,C 180,E1 -24997.713,E2 -24997.713} C_VEL
LIN {X 0,Y 129.142,Z 253.388,A -85,B 0,C 180,E1 -25000.941,E2 -25000.941} C_VEL
LIN {X 0,Y 129.393,Z 253.353,A -85,B 0,C 180,E1 -25007.819,E2 -25007.819} C_VEL
LIN {X 0,Y 129.483,Z 253.352,A -85,B 0,C 180,E1 -25010.628,E2 -25010.628} C_VEL
LIN {X 0,Y 130.048,Z 253.219,A -85,B 0,C 180,E1 -25019.999,E2 -25019.999} C_VEL
LIN {X 0,Y 129.442,Z 253.353,A -85,B 0,C 180,E1 -25029.373,E2 -25029.373} C_VEL
LIN {X 0,Y 129.273,Z 253.368,A -85,B 0,C 180,E1 -25032.559,E2 -25032.559} C_VEL
LIN {X 0,Y 129.058,Z 253.392,A -85,B 0,C 180,E1 -25039.07,E2 -25039.07} C_VEL
LIN {X 0,Y 129.02,Z 253.411,A -85,B 0,C 180,E1 -25042.413,E2 -25042.413} C_VEL
LIN {X 0,Y 128.996,Z 253.36,A -85,B 0,C 180,E1 -25049.362,E2 -25049.362} C_VEL
LIN {X 0,Y 128.934,Z 253.41,A -85,B 0,C 180,E1 -25055.169,E2 -25055.169} C_VEL
LIN {X 0,Y 128.903,Z 253.396,A -85,B 0,C 180,E1 -25060.862,E2 -25060.862} C_VEL
LIN {X 0,Y 128.895,Z 253.399,A -85,B 0,C 180,E1 -25065.138,E2 -25065.138} C_VEL
LIN {X 0,Y 128.948,Z 253.496,A -85,B 0,C 180,E1 -25070.442,E2 -25070.442} C_VEL
LIN {X 0,Y 129.945,Z 256.209,A -85,B 0,C 180,E1 -25071.151,E2 -25071.151} C_VEL
LIN {X 0,Y 132.226,Z 258.757,A -85,B 0,C 180,E1 -25072.417,E2 -25072.417} C_VEL
LIN {X 0,Y 134.449,Z 262.216,A -85,B 0,C 180,E1 -25073.659,E2 -25073.659} C_VEL
LIN {X 0,Y 136.05,Z 264.567,A -85,B 0,C 180,E1 -25074.509,E2 -25074.509} C_VEL
LIN {X 0,Y 140,Z 270.576,A -85,B 0,C 180,E1 -25076.491,E2 -25076.491} C_VEL
LIN {X 0,Y 146.444,Z 281.786,A -85,B 0,C 180,E1 -25079.471,E2 -25079.471} C_VEL
LIN {X 0,Y 153.045,Z 295.701,A -85,B 0,C 180,E1 -25082.293,E2 -25082.293} C_VEL
LIN {X 0,Y 153.973,Z 297.931,A -85,B 0,C 180,E1 -25082.678,E2 -25082.678} C_VEL
LIN {X 0,Y 150.711,Z 348.943,A -85,B 0,C 180,E1 -25084.841,E2 -25084.841} C_VEL
LIN {X 0,Y 149.136,Z 362.546,A -85,B 0,C 180,E1 -25085.933,E2 -25085.933} C_VEL
LIN {X 0,Y 147.073,Z 375.44,A -85,B 0,C 180,E1 -25087.532,E2 -25087.532} C_VEL
LIN {X 0,Y 144.645,Z 386.457,A -85,B 0,C 180,E1 -25089.381,E2 -25089.381} C_VEL
LIN {X 0,Y 141.955,Z 396.687,A -85,B 0,C 180,E1 -25091.609,E2 -25091.609} C_VEL
LIN {X 0,Y 138.938,Z 407.263,A -85,B 0,C 180,E1 -25094.606,E2 -25094.606} C_VEL
LIN {X 0,Y 135.824,Z 416.833,A -85,B 0,C 180,E1 -25098.061,E2 -25098.061} C_VEL
LIN {X 0,Y 132.634,Z 426.034,A -85,B 0,C 180,E1 -25102.394,E2 -25102.394} C_VEL
LIN {X 0,Y 130.141,Z 433.445,A -85,B 0,C 180,E1 -25106.91,E2 -25106.91} C_VEL
LIN {X 0,Y 128.375,Z 439.38,A -85,B 0,C 180,E1 -25111.574,E2 -25111.574} C_VEL
LIN {X 0,Y 127.133,Z 444.074,A -85,B 0,C 180,E1 -25116.353,E2 -25116.353} C_VEL
LIN {X 0,Y 126.38,Z 447.667,A -85,B 0,C 180,E1 -25121.228,E2 -25121.228} C_VEL
LIN {X 0,Y 126.276,Z 450.229,A -85,B 0,C 180,E1 -25126.162,E2 -25126.162} C_VEL
LIN {X 0,Y 126.593,Z 451.378,A -85,B 0,C 180,E1 -25129.461,E2 -25129.461} C_VEL
LIN {X 0,Y 127.187,Z 452.114,A -85,B 0,C 180,E1 -25132.759,E2 -25132.759} C_VEL
LIN {X 0,Y 128.111,Z 452.449,A -85,B 0,C 180,E1 -25136.035,E2 -25136.035} C_VEL
LIN {X 0,Y 129.69,Z 452.265,A -85,B 0,C 180,E1 -25139.884,E2 -25139.884} C_VEL
LIN {X 0,Y 132.965,Z 450.843,A -85,B 0,C 180,E1 -25145.553,E2 -25145.553} C_VEL
LIN {X 0,Y 135.716,Z 449.166,A -85,B 0,C 180,E1 -25149.036,E2 -25149.036} C_VEL
LIN {X 0,Y 140.935,Z 445.199,A -85,B 0,C 180,E1 -25154.28,E2 -25154.28} C_VEL
LIN {X 0,Y 145.814,Z 440.841,A -85,B 0,C 180,E1 -25158.132,E2 -25158.132} C_VEL
LIN {X 0,Y 151.645,Z 434.832,A -85,B 0,C 180,E1 -25161.987,E2 -25161.987} C_VEL
LIN {X 0,Y 157.864,Z 427.383,A -85,B 0,C 180,E1 -25165.448,E2 -25165.448} C_VEL
LIN {X 0,Y 164.613,Z 418.039,A -85,B 0,C 180,E1 -25168.636,E2 -25168.636} C_VEL
LIN {X 0,Y 170.646,Z 408.232,A -85,B 0,C 180,E1 -25171.064,E2 -25171.064} C_VEL
LIN {X 0,Y 176.271,Z 397.221,A -85,B 0,C 180,E1 -25173.137,E2 -25173.137} C_VEL
LIN {X 0,Y 180.675,Z 386.643,A -85,B 0,C 180,E1 -25174.667,E2 -25174.667} C_VEL
LIN {X 0,Y 184.649,Z 374.48,A -85,B 0,C 180,E1 -25175.987,E2 -25175.987} C_VEL
LIN {X 0,Y 187.783,Z 361.489,A -85,B 0,C 180,E1 -25176.997,E2 -25176.997} C_VEL
LIN {X 0,Y 189.767,Z 349.343,A -85,B 0,C 180,E1 -25177.618,E2 -25177.618} C_VEL
LIN {X 0,Y 191.454,Z 330.331,A -85,B 0,C 180,E1 -25178.253,E2 -25178.253} C_VEL
LIN {X 0,Y 186.863,Z 321.552,A -85,B 0,C 180,E1 -25181.57,E2 -25181.57} C_VEL
LIN {X 0,Y 183.396,Z 315.539,A -85,B 0,C 180,E1 -25184.441,E2 -25184.441} C_VEL
LIN {X 0,Y 181.148,Z 311.841,A -85,B 0,C 180,E1 -25186.54,E2 -25186.54} C_VEL
LIN {X 0,Y 178.98,Z 308.348,A -85,B 0,C 180,E1 -25188.821,E2 -25188.821} C_VEL
LIN {X 0,Y 177.111,Z 305.312,A -85,B 0,C 180,E1 -25191.081,E2 -25191.081} C_VEL
LIN {X 0,Y 174.836,Z 301.762,A -85,B 0,C 180,E1 -25194.446,E2 -25194.446} C_VEL
LIN {X 0,Y 174.143,Z 300.751,A -85,B 0,C 180,E1 -25195.678,E2 -25195.678} C_VEL
LIN {X 0,Y 172.315,Z 298.185,A -85,B 0,C 180,E1 -25199.863,E2 -25199.863} C_VEL
LIN {X 0,Y 171.746,Z 296.143,A -85,B 0,C 180,E1 -25202.346,E2 -25202.346} C_VEL
LIN {X 0,Y 171.583,Z 296.333,A -85,B 0,C 180,E1 -25211.507,E2 -25211.507} C_VEL
LIN {X 0,Y 173.133,Z 300.088,A -85,B 0,C 180,E1 -25216.85,E2 -25216.85} C_VEL
LIN {X 0,Y 174.643,Z 301.807,A -85,B 0,C 180,E1 -25219.71,E2 -25219.71} C_VEL
LIN {X 0,Y 177.889,Z 308.112,A -85,B 0,C 180,E1 -25224.513,E2 -25224.513} C_VEL
LIN {X 0,Y 180.787,Z 313.905,A -85,B 0,C 180,E1 -25227.808,E2 -25227.808} C_VEL
LIN {X 0,Y 183.928,Z 320.663,A -85,B 0,C 180,E1 -25230.848,E2 -25230.848} C_VEL
LIN {X 0,Y 187.236,Z 328.467,A -85,B 0,C 180,E1 -25233.668,E2 -25233.668} C_VEL
LIN {X 0,Y 190.51,Z 337.069,A -85,B 0,C 180,E1 -25236.175,E2 -25236.175} C_VEL
LIN {X 0,Y 190.936,Z 338.294,A -85,B 0,C 180,E1 -25236.487,E2 -25236.487} C_VEL
LIN {X 0,Y 188.827,Z 360.252,A -85,B 0,C 180,E1 -25237.202,E2 -25237.202} C_VEL
LIN {X 0,Y 186.41,Z 373.338,A -85,B 0,C 180,E1 -25237.867,E2 -25237.867} C_VEL
LIN {X 0,Y 183.231,Z 384.887,A -85,B 0,C 180,E1 -25238.682,E2 -25238.682} C_VEL
LIN {X 0,Y 178.765,Z 397.301,A -85,B 0,C 180,E1 -25239.948,E2 -25239.948} C_VEL
LIN {X 0,Y 173.625,Z 408.64,A -85,B 0,C 180,E1 -25241.51,E2 -25241.51} C_VEL
LIN {X 0,Y 168.091,Z 418.887,A -85,B 0,C 180,E1 -25243.409,E2 -25243.409} C_VEL
LIN {X 0,Y 162.765,Z 427.292,A -85,B 0,C 180,E1 -25245.439,E2 -25245.439} C_VEL
LIN {X 0,Y 156.12,Z 436.431,A -85,B 0,C 180,E1 -25248.394,E2 -25248.394} C_VEL
LIN {X 0,Y 150.003,Z 443.819,A -85,B 0,C 180,E1 -25251.624,E2 -25251.624} C_VEL
LIN {X 0,Y 143.621,Z 450.668,A -85,B 0,C 180,E1 -25255.752,E2 -25255.752} C_VEL
LIN {X 0,Y 138.922,Z 455.223,A -85,B 0,C 180,E1 -25259.606,E2 -25259.606} C_VEL
LIN {X 0,Y 134.818,Z 458.723,A -85,B 0,C 180,E1 -25263.695,E2 -25263.695} C_VEL
LIN {X 0,Y 131.499,Z 461.246,A -85,B 0,C 180,E1 -25268.027,E2 -25268.027} C_VEL
LIN {X 0,Y 129.69,Z 462.432,A -85,B 0,C 180,E1 -25271.022,E2 -25271.022} C_VEL
LIN {X 0,Y 127.44,Z 463.614,A -85,B 0,C 180,E1 -25277.252,E2 -25277.252} C_VEL
LIN {X 0,Y 126.552,Z 463.296,A -85,B 0,C 180,E1 -25283.618,E2 -25283.618} C_VEL
LIN {X 0,Y 126.662,Z 462.412,A -85,B 0,C 180,E1 -25287.156,E2 -25287.156} C_VEL
LIN {X 0,Y 126.754,Z 461.16,A -85,B 0,C 180,E1 -25290.354,E2 -25290.354} C_VEL
LIN {X 0,Y 126.606,Z 458.712,A -85,B 0,C 180,E1 -25294.77,E2 -25294.77} C_VEL
LIN {X 0,Y 126.896,Z 455.026,A -85,B 0,C 180,E1 -25299.558,E2 -25299.558} C_VEL
LIN {X 0,Y 127.485,Z 451.255,A -85,B 0,C 180,E1 -25303.355,E2 -25303.355} C_VEL
LIN {X 0,Y 127.462,Z 448.571,A -85,B 0,C 180,E1 -25305.714,E2 -25305.714} C_VEL
LIN {X 0,Y 126.071,Z 443.609,A -85,B 0,C 180,E1 -25309.56,E2 -25309.56} C_VEL
LIN {X 0,Y 125.091,Z 438.067,A -85,B 0,C 180,E1 -25313.299,E2 -25313.299} C_VEL
LIN {X 0,Y 125.692,Z 434.358,A -85,B 0,C 180,E1 -25315.392,E2 -25315.392} C_VEL
LIN {X 0,Y 127.567,Z 428.734,A -85,B 0,C 180,E1 -25318.104,E2 -25318.104} C_VEL
LIN {X 0,Y 130.464,Z 420.765,A -85,B 0,C 180,E1 -25321.222,E2 -25321.222} C_VEL
LIN {X 0,Y 133.783,Z 410.632,A -85,B 0,C 180,E1 -25324.373,E2 -25324.373} C_VEL
LIN {X 0,Y 137.1,Z 399.347,A -85,B 0,C 180,E1 -25327.026,E2 -25327.026} C_VEL
LIN {X 0,Y 140.281,Z 386.687,A -85,B 0,C 180,E1 -25329.225,E2 -25329.225} C_VEL
LIN {X 0,Y 142.677,Z 374.401,A -85,B 0,C 180,E1 -25330.732,E2 -25330.732} C_VEL
LIN {X 0,Y 144.471,Z 360.733,A -85,B 0,C 180,E1 -25331.853,E2 -25331.853} C_VEL
LIN {X 0,Y 147.011,Z 322.568,A -85,B 0,C 180,E1 -25333.565,E2 -25333.565} C_VEL
LIN {X 0,Y 146.955,Z 316.851,A -85,B 0,C 180,E1 -25333.93,E2 -25333.93} C_VEL
LIN {X 0,Y 145.882,Z 301.514,A -85,B 0,C 180,E1 -25335.204,E2 -25335.204} C_VEL
LIN {X 0,Y 141.725,Z 289.446,A -85,B 0,C 180,E1 -25337.345,E2 -25337.345} C_VEL
LIN {X 0,Y 136.443,Z 277.067,A -85,B 0,C 180,E1 -25340.156,E2 -25340.156} C_VEL
LIN {X 0,Y 133.577,Z 271.744,A -85,B 0,C 180,E1 -25341.731,E2 -25341.731} C_VEL
LIN {X 0,Y 127.954,Z 263.545,A -85,B 0,C 180,E1 -25344.956,E2 -25344.956} C_VEL
LIN {X 0,Y 125.717,Z 260.341,A -85,B 0,C 180,E1 -25346.371,E2 -25346.371} C_VEL
LIN {X 0,Y 125.1,Z 259.354,A -85,B 0,C 180,E1 -25346.786,E2 -25346.786} C_VEL
LIN {X 0,Y 122.923,Z 257.203,A -85,B 0,C 180,E1 -25348.191,E2 -25348.191} C_VEL
LIN {X 0,Y 121.895,Z 254.3,A -85,B 0,C 180,E1 -25349.124,E2 -25349.124} C_VEL
LIN {X 0,Y 121.924,Z 254.293,A -85,B 0,C 180,E1 -25352.538,E2 -25352.538} C_VEL
LIN {X 0,Y 122.01,Z 254.282,A -85,B 0,C 180,E1 -25357.138,E2 -25357.138} C_VEL
LIN {X 0,Y 122.092,Z 254.27,A -85,B 0,C 180,E1 -25363.272,E2 -25363.272} C_VEL
LIN {X 0,Y 122.34,Z 254.233,A -85,B 0,C 180,E1 -25367.527,E2 -25367.527} C_VEL
LIN {X 0,Y 122.416,Z 254.227,A -85,B 0,C 180,E1 -25370.081,E2 -25370.081} C_VEL
LIN {X 0,Y 122.566,Z 254.168,A -85,B 0,C 180,E1 -25376.712,E2 -25376.712} C_VEL
LIN {X 0,Y 123.001,Z 254.095,A -85,B 0,C 180,E1 -25379.999,E2 -25379.999} C_VEL
LIN {X 0,Y 122.358,Z 254.236,A -85,B 0,C 180,E1 -25387.104,E2 -25387.104} C_VEL
LIN {X 0,Y 122.263,Z 254.239,A -85,B 0,C 180,E1 -25392.308,E2 -25392.308} C_VEL
LIN {X 0,Y 122.035,Z 254.28,A -85,B 0,C 180,E1 -25396.734,E2 -25396.734} C_VEL
LIN {X 0,Y 121.963,Z 254.292,A -85,B 0,C 180,E1 -25402.809,E2 -25402.809} C_VEL
LIN {X 0,Y 121.905,Z 254.237,A -85,B 0,C 180,E1 -25410.164,E2 -25410.164} C_VEL
LIN {X 0,Y 121.859,Z 254.3,A -85,B 0,C 180,E1 -25416.172,E2 -25416.172} C_VEL
LIN {X 0,Y 121.827,Z 254.271,A -85,B 0,C 180,E1 -25421.429,E2 -25421.429} C_VEL
LIN {X 0,Y 121.82,Z 254.459,A -85,B 0,C 180,E1 -25426.651,E2 -25426.651} C_VEL
LIN {X 0,Y 122.737,Z 257.032,A -85,B 0,C 180,E1 -25427.434,E2 -25427.434} C_VEL
LIN {X 0,Y 124.816,Z 259.241,A -85,B 0,C 180,E1 -25428.799,E2 -25428.799} C_VEL
LIN {X 0,Y 125.573,Z 260.083,A -85,B 0,C 180,E1 -25429.279,E2 -25429.279} C_VEL
LIN {X 0,Y 127.656,Z 263.247,A -85,B 0,C 180,E1 -25430.619,E2 -25430.619} C_VEL
LIN {X 0,Y 129.04,Z 265.156,A -85,B 0,C 180,E1 -25431.452,E2 -25431.452} C_VEL
LIN {X 0,Y 133.874,Z 272.242,A -85,B 0,C 180,E1 -25434.17,E2 -25434.17} C_VEL
LIN {X 0,Y 140.17,Z 283.064,A -85,B 0,C 180,E1 -25437.413,E2 -25437.413} C_VEL
LIN {X 0,Y 146.043,Z 295.013,A -85,B 0,C 180,E1 -25440.178,E2 -25440.178} C_VEL
LIN {X 0,Y 148.125,Z 299.788,A -85,B 0,C 180,E1 -25441.114,E2 -25441.114} C_VEL
LIN {X 0,Y 144.856,Z 349.42,A -85,B 0,C 180,E1 -25443.292,E2 -25443.292} C_VEL
LIN {X 0,Y 143.24,Z 362.739,A -85,B 0,C 180,E1 -25444.389,E2 -25444.389} C_VEL
LIN {X 0,Y 141.162,Z 375.161,A -85,B 0,C 180,E1 -25445.952,E2 -25445.952} C_VEL
LIN {X 0,Y 138.409,Z 387.112,A -85,B 0,C 180,E1 -25448.015,E2 -25448.015} C_VEL
LIN {X 0,Y 135.242,Z 398.57,A -85,B 0,C 180,E1 -25450.661,E2 -25450.661} C_VEL
LIN {X 0,Y 132.347,Z 408.001,A -85,B 0,C 180,E1 -25453.491,E2 -25453.491} C_VEL
LIN {X 0,Y 129.534,Z 416.268,A -85,B 0,C 180,E1 -25456.595,E2 -25456.595} C_VEL
LIN {X 0,Y 126.579,Z 424.417,A -85,B 0,C 180,E1 -25460.418,E2 -25460.418} C_VEL
LIN {X 0,Y 123.793,Z 432.185,A -85,B 0,C 180,E1 -25465.121,E2 -25465.121} C_VEL
LIN {X 0,Y 121.732,Z 438.42,A -85,B 0,C 180,E1 -25470.006,E2 -25470.006} C_VEL
LIN {X 0,Y 120.416,Z 443.024,A -85,B 0,C 180,E1 -25474.619,E2 -25474.619} C_VEL
LIN {X 0,Y 119.387,Z 447.227,A -85,B 0,C 180,E1 -25480.177,E2 -25480.177} C_VEL
LIN {X 0,Y 119.123,Z 449.224,A -85,B 0,C 180,E1 -25483.655,E2 -25483.655} C_VEL
LIN {X 0,Y 119.53,Z 451.64,A -85,B 0,C 180,E1 -25489.825,E2 -25489.825} C_VEL
LIN {X 0,Y 120.403,Z 452.529,A -85,B 0,C 180,E1 -25494.121,E2 -25494.121} C_VEL
LIN {X 0,Y 121.481,Z 452.807,A -85,B 0,C 180,E1 -25497.573,E2 -25497.573} C_VEL
LIN {X 0,Y 122.982,Z 452.612,A -85,B 0,C 180,E1 -25500.999,E2 -25500.999} C_VEL
LIN {X 0,Y 124.783,Z 452.018,A -85,B 0,C 180,E1 -25504.282,E2 -25504.282} C_VEL
LIN {X 0,Y 126.975,Z 451.007,A -85,B 0,C 180,E1 -25507.509,E2 -25507.509} C_VEL
LIN {X 0,Y 129.556,Z 449.516,A -85,B 0,C 180,E1 -25510.617,E2 -25510.617} C_VEL
LIN {X 0,Y 134.039,Z 446.414,A -85,B 0,C 180,E1 -25515.062,E2 -25515.062} C_VEL
LIN {X 0,Y 139.25,Z 442.161,A -85,B 0,C 180,E1 -25519.207,E2 -25519.207} C_VEL
LIN {X 0,Y 145.1,Z 436.624,A -85,B 0,C 180,E1 -25523.053,E2 -25523.053} C_VEL
LIN {X 0,Y 151.484,Z 429.608,A -85,B 0,C 180,E1 -25526.627,E2 -25526.627} C_VEL
LIN {X 0,Y 157.268,Z 422.375,A -85,B 0,C 180,E1 -25529.344,E2 -25529.344} C_VEL
LIN {X 0,Y 162.944,Z 414.252,A -85,B 0,C 180,E1 -25531.678,E2 -25531.678} C_VEL
LIN {X 0,Y 169.117,Z 403.721,A -85,B 0,C 180,E1 -25533.983,E2 -25533.983} C_VEL
LIN {X 0,Y 174.365,Z 392.906,A -85,B 0,C 180,E1 -25535.771,E2 -25535.771} C_VEL
LIN {X 0,Y 178.763,Z 381.631,A -85,B 0,C 180,E1 -25537.207,E2 -25537.207} C_VEL
LIN {X 0,Y 182.335,Z 369.847,A -85,B 0,C 180,E1 -25538.296,E2 -25538.296} C_VEL
LIN {X 0,Y 185.15,Z 356.651,A -85,B 0,C 180,E1 -25539.181,E2 -25539.181} C_VEL
LIN {X 0,Y 186.945,Z 343.247,A -85,B 0,C 180,E1 -25539.702,E2 -25539.702} C_VEL
LIN {X 0,Y 187.727,Z 333.866,A -85,B 0,C 180,E1 -25540.017,E2 -25540.017} C_VEL
LIN {X 0,Y 183.25,Z 325.033,A -85,B 0,C 180,E1 -25543.625,E2 -25543.625} C_VEL
LIN {X 0,Y 179.503,Z 318.533,A -85,B 0,C 180,E1 -25547.159,E2 -25547.159} C_VEL
LIN {X 0,Y 177.322,Z 314.85,A -85,B 0,C 180,E1 -25549.583,E2 -25549.583} C_VEL
LIN {X 0,Y 175.539,Z 311.87,A -85,B 0,C 180,E1 -25551.873,E2 -25551.873} C_VEL
LIN {X 0,Y 173.081,Z 307.694,A -85,B 0,C 180,E1 -25555.96,E2 -25555.96} C_VEL
LIN {X 0,Y 171.264,Z 305.109,A -85,B 0,C 180,E1 -25560.321,E2 -25560.321} C_VEL
LIN {X 0,Y 170.841,Z 303.316,A -85,B 0,C 180,E1 -25562.358,E2 -25562.358} C_VEL
LIN {X 0,Y 170.513,Z 303.237,A -85,B 0,C 180,E1 -25570.533,E2 -25570.533} C_VEL
LIN {X 0,Y 170.694,Z 303.835,A -85,B 0,C 180,E1 -25571.724,E2 -25571.724} C_VEL
LIN {X 0,Y 172.581,Z 307.604,A -85,B 0,C 180,E1 -25577.593,E2 -25577.593} C_VEL
LIN {X 0,Y 173.467,Z 308.768,A -85,B 0,C 180,E1 -25579.287,E2 -25579.287} C_VEL
LIN {X 0,Y 176.334,Z 314.698,A -85,B 0,C 180,E1 -25583.808,E2 -25583.808} C_VEL
LIN {X 0,Y 179.096,Z 320.577,A -85,B 0,C 180,E1 -25587.142,E2 -25587.142} C_VEL
LIN {X 0,Y 182.406,Z 328.333,A -85,B 0,C 180,E1 -25590.518,E2 -25590.518} C_VEL
LIN {X 0,Y 185.418,Z 336.028,A -85,B 0,C 180,E1 -25593.208,E2 -25593.208} C_VEL
LIN {X 0,Y 187.182,Z 341.031,A -85,B 0,C 180,E1 -25594.675,E2 -25594.675} C_VEL
LIN {X 0,Y 185.17,Z 360.775,A -85,B 0,C 180,E1 -25595.346,E2 -25595.346} C_VEL
LIN {X 0,Y 182.516,Z 374.261,A -85,B 0,C 180,E1 -25596.039,E2 -25596.039} C_VEL
LIN {X 0,Y 179.031,Z 386.072,A -85,B 0,C 180,E1 -25596.893,E2 -25596.893} C_VEL
LIN {X 0,Y 174.318,Z 398.405,A -85,B 0,C 180,E1 -25598.17,E2 -25598.17} C_VEL
LIN {X 0,Y 169.023,Z 409.482,A -85,B 0,C 180,E1 -25599.715,E2 -25599.715} C_VEL
LIN {X 0,Y 163.947,Z 418.464,A -85,B 0,C 180,E1 -25601.394,E2 -25601.394} C_VEL
LIN {X 0,Y 157.795,Z 427.721,A -85,B 0,C 180,E1 -25603.634,E2 -25603.634} C_VEL
LIN {X 0,Y 150.905,Z 436.718,A -85,B 0,C 180,E1 -25606.61,E2 -25606.61} C_VEL
LIN {X 0,Y 144.496,Z 443.999,A -85,B 0,C 180,E1 -25609.873,E2 -25609.873} C_VEL
LIN {X 0,Y 137.785,Z 450.707,A -85,B 0,C 180,E1 -25614.083,E2 -25614.083} C_VEL
LIN {X 0,Y 132.83,Z 455.178,A -85,B 0,C 180,E1 -25618.053,E2 -25618.053} C_VEL
LIN {X 0,Y 129.897,Z 457.558,A -85,B 0,C 180,E1 -25620.857,E2 -25620.857} C_VEL
LIN {X 0,Y 127.18,Z 459.52,A -85,B 0,C 180,E1 -25623.76,E2 -25623.76} C_VEL
LIN {X 0,Y 124.923,Z 461.076,A -85,B 0,C 180,E1 -25626.804,E2 -25626.804} C_VEL
LIN {X 0,Y 121.537,Z 462.935,A -85,B 0,C 180,E1 -25633.19,E2 -25633.19} C_VEL
LIN {X 0,Y 119.818,Z 463.298,A -85,B 0,C 180,E1 -25639.86,E2 -25639.86} C_VEL
LIN {X 0,Y 119.505,Z 462.886,A -85,B 0,C 180,E1 -25643.24,E2 -25643.24} C_VEL
LIN {X 0,Y 119.587,Z 461.779,A -85,B 0,C 180,E1 -25647.551,E2 -25647.551} C_VEL
LIN {X 0,Y 119.695,Z 460.847,A -85,B 0,C 180,E1 -25649.994,E2 -25649.994} C_VEL
LIN {X 0,Y 119.528,Z 458.141,A -85,B 0,C 180,E1 -25655.054,E2 -25655.054} C_VEL
LIN {X 0,Y 119.857,Z 454.368,A -85,B 0,C 180,E1 -25660.125,E2 -25660.125} C_VEL
LIN {X 0,Y 120.797,Z 449.426,A -85,B 0,C 180,E1 -25665.17,E2 -25665.17} C_VEL
LIN {X 0,Y 122.722,Z 443.196,A -85,B 0,C 180,E1 -25670.089,E2 -25670.089} C_VEL
LIN {X 0,Y 125.353,Z 435.396,A -85,B 0,C 180,E1 -25674.857,E2 -25674.857} C_VEL
LIN {X 0,Y 125.692,Z 434.358,A -85,B 0,C 180,E1 -25675.392,E2 -25675.392} C_VEL
LIN {X 0,Y 126.4,Z 430.505,A -85,B 0,C 180,E1 -25677.383,E2 -25677.383} C_VEL
LIN {X 0,Y 126.137,Z 423.812,A -85,B 0,C 180,E1 -25680.688,E2 -25680.688} C_VEL
LIN {X 0,Y 126.042,Z 416.611,A -85,B 0,C 180,E1 -25683.796,E2 -25683.796} C_VEL
LIN {X 0,Y 126.977,Z 411.905,A -85,B 0,C 180,E1 -25685.405,E2 -25685.405} C_VEL
LIN {X 0,Y 130.507,Z 400.745,A -85,B 0,C 180,E1 -25688.253,E2 -25688.253} C_VEL
LIN {X 0,Y 132.854,Z 392.374,A -85,B 0,C 180,E1 -25689.886,E2 -25689.886} C_VEL
LIN {X 0,Y 135.532,Z 380.925,A -85,B 0,C 180,E1 -25691.624,E2 -25691.624} C_VEL
LIN {X 0,Y 137.779,Z 368.103,A -85,B 0,C 180,E1 -25692.979,E2 -25692.979} C_VEL
LIN {X 0,Y 139.285,Z 354.62,A -85,B 0,C 180,E1 -25693.866,E2 -25693.866} C_VEL
LIN {X 0,Y 141.443,Z 320.138,A -85,B 0,C 180,E1 -25695.425,E2 -25695.425} C_VEL
LIN {X 0,Y 140.506,Z 303.965,A -85,B 0,C 180,E1 -25696.798,E2 -25696.798} C_VEL
LIN {X 0,Y 136.594,Z 292.379,A -85,B 0,C 180,E1 -25699.003,E2 -25699.003} C_VEL
LIN {X 0,Y 131.651,Z 280.607,A -85,B 0,C 180,E1 -25701.883,E2 -25701.883} C_VEL
LIN {X 0,Y 129.018,Z 275.974,A -85,B 0,C 180,E1 -25703.429,E2 -25703.429} C_VEL
LIN {X 0,Y 124.243,Z 268.811,A -85,B 0,C 180,E1 -25706.406,E2 -25706.406} C_VEL
LIN {X 0,Y 121.53,Z 264.947,A -85,B 0,C 180,E1 -25708.271,E2 -25708.271} C_VEL
LIN {X 0,Y 119.166,Z 261.892,A -85,B 0,C 180,E1 -25710.002,E2 -25710.002} C_VEL
LIN {X 0,Y 118.428,Z 260.483,A -85,B 0,C 180,E1 -25710.617,E2 -25710.617} C_VEL
LIN {X 0,Y 116.243,Z 258.524,A -85,B 0,C 180,E1 -25712.303,E2 -25712.303} C_VEL
LIN {X 0,Y 115.108,Z 256.381,A -85,B 0,C 180,E1 -25713.359,E2 -25713.359} C_VEL
LIN {X 0,Y 114.859,Z 255.177,A -85,B 0,C 180,E1 -25713.786,E2 -25713.786} C_VEL
LIN {X 0,Y 114.967,Z 255.165,A -85,B 0,C 180,E1 -25718.481,E2 -25718.481} C_VEL
LIN {X 0,Y 115.125,Z 255.143,A -85,B 0,C 180,E1 -25725.865,E2 -25725.865} C_VEL
LIN {X 0,Y 115.336,Z 255.105,A -85,B 0,C 180,E1 -25729.466,E2 -25729.466} C_VEL
LIN {X 0,Y 115.492,Z 255.048,A -85,B 0,C 180,E1 -25736.51,E2 -25736.51} C_VEL
LIN {X 0,Y 115.928,Z 254.973,A -85,B 0,C 180,E1 -25739.999,E2 -25739.999} C_VEL
LIN {X 0,Y 115.329,Z 255.118,A -85,B 0,C 180,E1 -25746.999,E2 -25746.999} C_VEL
LIN {X 0,Y 115.18,Z 255.122,A -85,B 0,C 180,E1 -25752.556,E2 -25752.556} C_VEL
LIN {X 0,Y 114.94,Z 255.155,A -85,B 0,C 180,E1 -25757.801,E2 -25757.801} C_VEL
LIN {X 0,Y 114.884,Z 255.174,A -85,B 0,C 180,E1 -25763.446,E2 -25763.446} C_VEL
LIN {X 0,Y 114.832,Z 255.116,A -85,B 0,C 180,E1 -25771.058,E2 -25771.058} C_VEL
LIN {X 0,Y 114.755,Z 255.188,A -85,B 0,C 180,E1 -25777.764,E2 -25777.764} C_VEL
LIN {X 0,Y 114.756,Z 255.147,A -85,B 0,C 180,E1 -25781.98,E2 -25781.98} C_VEL
